// TwinCAT 3 PLC project Untitled1
// ProgramVersion: 3.1.0.8
// libraries:
//   Indradrive Library, * (Bosch)
//   Recipe Management, 3.3.1.0 (System)
//   Standard, * (System)
//   VisuElem3DPath, 3.5.6.0 (System)
//   VisuElemMeter, 3.5.6.0 (System)
//   VisuElems, 3.5.6.10 (System)
//   VisuElemsDateTime, 3.5.6.0 (System)
//   VisuElemsSpecialControls, 3.5.6.0 (System)
//   VisuElemsWinControls, 3.5.6.0 (System)
//   VisuElemTextEditor, 3.5.6.0 (System)
//   visuinputs, 3.5.6.0 (system)
//   VisuNativeControl, 3.5.6.0 (System)
//   Tc2_IoFunctions, * (Beckhoff Automation GmbH)
//   Tc2_Standard, * (Beckhoff Automation GmbH)
//   Tc2_System, * (Beckhoff Automation GmbH)
//   Tc2_Utilities, * (Beckhoff Automation GmbH)
//   Tc3_Interfaces, * (Beckhoff Automation GmbH)
//   Tc3_Module, * (Beckhoff Automation GmbH)
// project tree:
//   DUTs/ structCylinder.TcDUT, structHBMSerialCtrl.TcDUT, structHMI.TcDUT, structIndradrive.TcDUT, structMachineCtrl.TcDUT, structMachineData.TcDUT, structMotorDirect.TcDUT, structMotorInverter.TcDUT, structRecipe.TcDUT, structStationCtrl.TcDUT, structStatistic.TcDUT, structVacuum.TcDUT
//   / GlobalTextList.TcGTLO, PlcTask.TcTTO, RecipeManager.TcRMO (not stored), Visualization Manager.TcVMO (not stored)
//   GVLs/Device/ GVL_Cylinder.TcGVL, GVL_Motor.TcGVL, GVL_Nordson.TcGVL, GVL_Servo.TcGVL, GVL_Vacuum.TcGVL
//   GVLs/IO/ GVL_Ethercat.TcGVL, GVL_IO_CO.TcGVL, GVL_IO_EL.TcGVL, GVL_IO_HOR.TcGVL, GVL_IO_ER.TcGVL, GVL_Valve_Manifold.TcGVL
//   GVLs/MC/ GVL_General.TcGVL, GVL_Auto.TcGVL, GVL_Holding.TcGVL, GVL_Origin.TcGVL, GVL_Error.TcGVL, GVL_Configuration.TcGVL, GVL_HMI.TcGVL, GVL_Status.TcGVL, GVL_Symbol_Spec.TcGVL, GVL_Timer.TcGVL
//   POUs/Collator/ CO_Cylinder_Output.TcPOU, CO_Main.TcPOU, CO_Nordson.TcPOU, CO_Servo_Output.TcPOU, CO_Motor_Output.TcPOU, CO_Timers.TcPOU, CO_TestServo.TcPOU
//   POUs/Collator/Y Pusher n Bridge/ CO_YPush_Auto.TcPOU, CO_YPush_Error.TcPOU, CO_YPush_Origin.TcPOU
//   POUs/Erector/ ER_Auto_Arm.TcPOU, ER_Auto_FixedFlap.TcPOU, ER_Error.TcPOU, ER_Glue.TcPOU, ER_Origin.TcPOU, ER_Cylinder_Output.TcPOU, ER_Main.TcPOU, ER_Motor_Output.TcPOU, ER_Servo_Output.TcPOU, ER_Timers.TcPOU, ER_Vacuum_Output.TcPOU
//   POUs/Exit/ EX_Auto.TcPOU, EX_Error.TcPOU, EX_Origin.TcPOU, EX_Main.TcPOU, EX_Motor_Output.TcPOU, EX_Cylinder_Output.TcPOU, EX_LoadCell_Output.TcPOU, EX_Servo_Output.TcPOU
//   POUs/FastTask/ CO_StkRel_Cyl_FastOutput.TcPOU, FastTask_Main.TcPOU
//   POUs/FB/ fbCalculateTotalTime.TcPOU, fbCylinderCtrl_2Station.TcPOU, fbCylinderCtrl.TcPOU, fbIndradrive.TcPOU, fbMachineCtrl.TcPOU, fbMotorInverterCtrl.TcPOU, fbVacuumPumpCtrl.TcPOU, fbOnOffDevCtrl.TcPOU, fbMotorDirectCtrl.TcPOU, fbVacuumValveCtrl.TcPOU, fcComparePos.TcPOU, fcCompareWAPos.TcPOU
//   POUs/Horizontal/ Downstream_Conveyor.TcPOU, HOR_Servo_Output.TcPOU, HOR_Auto.TcPOU, HOR_Error.TcPOU, HOR_Main.TcPOU, HOR_Motor_Output.TcPOU, HOR_Origin.TcPOU, HOR_Timers.TcPOU, Option_90Deg_Conv.TcPOU
//   POUs/MC/ Calc_McPerformance.TcPOU, Check_AutorunCond.TcPOU, Check_Ethercat.TcPOU, Guard_Door.TcPOU, Emergency_Stop.TcPOU, MAIN.TcPOU, Memory_Handling.TcPOU, Recipe_Handling.TcPOU, Statistic.TcPOU, Std_System_Out.TcPOU, TouchScreen.TcPOU, Track_and_Trace.TcPOU, WarningMsg.TcPOU
//   VISUs/FB/ Std_Cylinder_Ctrl.TcVIS, Std_OnOffDev_Ctrl.TcVIS, Std_VacuumVal_Ctrl.TcVIS, Std_BoschServo_Ctrl.TcVIS
//   VISUs/Obj_Button/ ButtonGreenInd.TcVIS
//   VISUs/Obj_Indicator/ Blue_Ind.TcVIS, Green_Ind.TcVIS, Red_Ind.TcVIS, Yellow_Ind.TcVIS
//   VISUs/Obj_Switch/ ToggleSwitch1.TcVIS
//   VISUs/Prog/ IO_Monitor.TcVIS, MANUAL_STEP.TcVIS, resetbtn.TcVIS, Std_NewPassWord.TcVIS, Std_Password.TcVIS
// real-time tasks:
//   TASK PlcTask: cycle T#10ms, priority 20, ADS port 350
// I/O:
//   DEVICE Device 1 (EtherCAT), AmsNetId 169.254.27.43.2.1
//     EractorRemoteIO (EK1101) [EK1101 EtherCAT Coupler (2A E-Bus, ID switch)]
//       41DI1 (EL1809) [EL1809 16Ch. Dig. Input 24V, 3ms]
//       41DI2 (EL1809) [EL1809 16Ch. Dig. Input 24V, 3ms]
//       41DO1 (EL2809) [EL2809 16Ch. Dig. Output 24V, 0.5A]
//       41DO2 (EL2809) [EL2809 16Ch. Dig. Output 24V, 0.5A]
//       41PO1 (EL9510) [EL9510 Power supply terminal 10V] (disabled)
//       41AI1 (EL3356) [EL3356 1Ch. Ana. Input Resistor Bridge Terminal, 16bit, High Precision] (disabled)
//       41BC2 (EK1122) [EK1122 2 port EtherCAT junction]
//         EractorArmLeftValveBlock (CTEU-EtherCAT 16Byte) [CTEU-EtherCAT Fieldbus module 16Byte fix]
//         60A1 (EP1008-0001) [EP1008-0001 8 Ch. Dig. Input 24V, 3ms, M8]
//         61A1 (EP1008-0001) [EP1008-0001 8 Ch. Dig. Input 24V, 3ms, M8]
//         62A1 (EP1008-0001) [EP1008-0001 8 Ch. Dig. Input 24V, 3ms, M8]
//         66A1 (EP1008-0001) [EP1008-0001 8 Ch. Dig. Input 24V, 3ms, M8]
//         EractorArm (IndraDrive MPB16/17) [IndraDrive MPB16/17]
//         Eractor Main WA (IndraDrive MPB16/17) [IndraDrive MPB16/17]
//         Eractor HeightL WA (IndraDrive MPB16/17) [IndraDrive MPB16/17]
//         Eractor HeightR WA (IndraDrive MPB16/17) [IndraDrive MPB16/17]
//       41BC3 (EK1122) [EK1122 2 port EtherCAT junction]
//         241BC1 CollactorRemoteIO (EK1101) [EK1101 EtherCAT Coupler (2A E-Bus, ID switch)]
//           241DI1 (EL1809) [EL1809 16Ch. Dig. Input 24V, 3ms]
//           241DI2 (EL1809) [EL1809 16Ch. Dig. Input 24V, 3ms]
//           241DO1 (EL2809) [EL2809 16Ch. Dig. Output 24V, 0.5A]
//           241DO2 (EL2809) [EL2809 16Ch. Dig. Output 24V, 0.5A]
//           241BC2 (EK1122) [EK1122 2 port EtherCAT junction]
//             270A1 (CTEU-EtherCAT 16Byte) [CTEU-EtherCAT Fieldbus module 16Byte fix]
//             263A1 (EP1008-0001) [EP1008-0001 8 Ch. Dig. Input 24V, 3ms, M8]
//             264A1 (EP1008-0001) [EP1008-0001 8 Ch. Dig. Input 24V, 3ms, M8]
//             262A1 (EP1008-0001) [EP1008-0001 8 Ch. Dig. Input 24V, 3ms, M8]
//             265A1 (EP1008-0001) [EP1008-0001 8 Ch. Dig. Input 24V, 3ms, M8]
//             Tilter (IndraDrive MPB16/17) [IndraDrive MPB16/17]
//             YPusher (IndraDrive MPB16/17) [IndraDrive MPB16/17]
//         260A1 (EP1008-0001) [EP1008-0001 8 Ch. Dig. Input 24V, 3ms, M8]
//     EractorArmRightValveBlock (CTEU-EtherCAT 16Byte) [CTEU-EtherCAT Fieldbus module 16Byte fix]
//     63A1 (EP1008-0001) [EP1008-0001 8 Ch. Dig. Input 24V, 3ms, M8]
//     64A1 (EP1008-0001) [EP1008-0001 8 Ch. Dig. Input 24V, 3ms, M8]
//     65A1 (EP1008-0001) [EP1008-0001 8 Ch. Dig. Input 24V, 3ms, M8]
// variable links:
//   Untitled1/Untitled1 Instance <-> Device 1 (EtherCAT)/63A1 (EP1008-0001)
//     PlcTask Inputs/GVL_Ethercat.I_ECat_63A1 <-> InfoData/State
//     PlcTask Inputs/GVL_IO_ER.I_ER_BFlapR_Bwd <-> Channel 8/Input
//     PlcTask Inputs/GVL_IO_ER.I_ER_BFlapR_Fwd <-> Channel 7/Input
//     PlcTask Inputs/GVL_IO_ER.I_ER_BufferR_PE <-> Channel 1/Input
//     PlcTask Inputs/GVL_IO_ER.I_ER_EmptyR_PE <-> Channel 2/Input
//     PlcTask Inputs/GVL_IO_ER.I_ER_FFlapR_Bwd <-> Channel 6/Input
//     PlcTask Inputs/GVL_IO_ER.I_ER_FFlapR_Fwd <-> Channel 5/Input
//     PlcTask Inputs/GVL_IO_ER.I_EX_StpR_Dn <-> Channel 4/Input
//   Untitled1/Untitled1 Instance <-> Device 1 (EtherCAT)/64A1 (EP1008-0001)
//     PlcTask Inputs/GVL_Ethercat.I_ECat_64A1 <-> InfoData/State
//     PlcTask Inputs/GVL_IO_ER.I_ER_BFlapR_VacSw <-> Channel 7/Input
//     PlcTask Inputs/GVL_IO_ER.I_ER_CaseGuideR_Bwd <-> Channel 4/Input
//     PlcTask Inputs/GVL_IO_ER.I_ER_CaseGuideR_Fwd <-> Channel 3/Input
//     PlcTask Inputs/GVL_IO_ER.I_ER_RFlapR_Bwd <-> Channel 6/Input
//     PlcTask Inputs/GVL_IO_ER.I_ER_RFlapR_Fwd <-> Channel 5/Input
//     PlcTask Inputs/GVL_IO_ER.I_ER_StpR_Ctn_PE <-> Channel 8/Input
//     PlcTask Inputs/GVL_IO_ER.I_ER_StpR_Dn <-> Channel 2/Input
//     PlcTask Inputs/GVL_IO_ER.I_ER_StpR_Up <-> Channel 1/Input
//   Untitled1/Untitled1 Instance <-> Device 1 (EtherCAT)/65A1 (EP1008-0001)
//     PlcTask Inputs/GVL_Ethercat.I_ECat_65A1 <-> InfoData/State
//     PlcTask Inputs/GVL_IO_ER.I_ER_FlapHoldR_Bwd <-> Channel 6/Input
//     PlcTask Inputs/GVL_IO_ER.I_ER_FlapHoldR_Fwd <-> Channel 5/Input
//     PlcTask Inputs/GVL_IO_ER.I_ER_TFlapClsR_Bwd <-> Channel 4/Input
//     PlcTask Inputs/GVL_IO_ER.I_ER_TFlapClsR_Fwd <-> Channel 3/Input
//     PlcTask Inputs/GVL_IO_ER.I_ER_TFlapOpnR_Bwd <-> Channel 2/Input
//     PlcTask Inputs/GVL_IO_ER.I_ER_TFlapOpnR_Fwd <-> Channel 1/Input
//     PlcTask Inputs/GVL_IO_ER.I_EX_SquarenessR_Bwd <-> Channel 8/Input
//     PlcTask Inputs/GVL_IO_ER.I_EX_SquarenessR_Fwd <-> Channel 7/Input
//   Untitled1/Untitled1 Instance <-> Device 1 (EtherCAT)/EractorArmRightValveBlock (CTEU-EtherCAT 16Byte)
//     PlcTask Inputs/GVL_Ethercat.I_ECat_71A1 <-> InfoData/State
//     PlcTask Outputs/GVL_Valve_Manifold.QW_71A1_{1..4} <-> Outputs/QB{0..3}  (4 links)
//   Untitled1/Untitled1 Instance <-> Device 1 (EtherCAT)/EractorRemoteIO (EK1101)
//     PlcTask Inputs/GVL_Ethercat.I_ECat_41BC1 <-> InfoData/State
//   Untitled1/Untitled1 Instance <-> Device 1 (EtherCAT)/EractorRemoteIO (EK1101)/41AI1 (EL3356)
//     PlcTask Inputs/GVL_IO_ER.I_Weighing <-> RMB Value (INT32)/Value
//     PlcTask Inputs/GVL_IO_ER.I_Weighing_Status_SteadyBit <-> RMB Status/Status/Steady state
//   Untitled1/Untitled1 Instance <-> Device 1 (EtherCAT)/EractorRemoteIO (EK1101)/41BC2 (EK1122)
//     PlcTask Inputs/GVL_Ethercat.I_ECat_41BC2 <-> InfoData/State
//   Untitled1/Untitled1 Instance <-> Device 1 (EtherCAT)/EractorRemoteIO (EK1101)/41BC2 (EK1122)/60A1 (EP1008-0001)
//     PlcTask Inputs/GVL_Ethercat.I_ECat_60A1 <-> InfoData/State
//     PlcTask Inputs/GVL_IO_ER.I_ER_BFlapL_Bwd <-> Channel 8/Input
//     PlcTask Inputs/GVL_IO_ER.I_ER_BFlapL_Fwd <-> Channel 7/Input
//     PlcTask Inputs/GVL_IO_ER.I_ER_BufferL_PE <-> Channel 1/Input
//     PlcTask Inputs/GVL_IO_ER.I_ER_EmptyL_PE <-> Channel 2/Input
//     PlcTask Inputs/GVL_IO_ER.I_ER_FFlapL_Bwd <-> Channel 6/Input
//     PlcTask Inputs/GVL_IO_ER.I_ER_FFlapL_Fwd <-> Channel 5/Input
//     PlcTask Inputs/GVL_IO_ER.I_ER_RefillL_PE <-> Channel 3/Input
//     PlcTask Inputs/GVL_IO_ER.I_EX_StpL_Dn <-> Channel 4/Input
//   Untitled1/Untitled1 Instance <-> Device 1 (EtherCAT)/EractorRemoteIO (EK1101)/41BC2 (EK1122)/61A1 (EP1008-0001)
//     PlcTask Inputs/GVL_Ethercat.I_ECat_61A1 <-> InfoData/State
//     PlcTask Inputs/GVL_IO_ER.I_ER_BFlapL_VacSw <-> Channel 7/Input
//     PlcTask Inputs/GVL_IO_ER.I_ER_CaseGuideL_Bwd <-> Channel 4/Input
//     PlcTask Inputs/GVL_IO_ER.I_ER_CaseGuideL_Fwd <-> Channel 3/Input
//     PlcTask Inputs/GVL_IO_ER.I_ER_RFlapL_Bwd <-> Channel 6/Input
//     PlcTask Inputs/GVL_IO_ER.I_ER_RFlapL_Fwd <-> Channel 5/Input
//     PlcTask Inputs/GVL_IO_ER.I_ER_StpL_Ctn_PE <-> Channel 8/Input
//     PlcTask Inputs/GVL_IO_ER.I_ER_StpL_Dn <-> Channel 2/Input
//     PlcTask Inputs/GVL_IO_ER.I_ER_StpL_Up <-> Channel 1/Input
//   Untitled1/Untitled1 Instance <-> Device 1 (EtherCAT)/EractorRemoteIO (EK1101)/41BC2 (EK1122)/62A1 (EP1008-0001)
//     PlcTask Inputs/GVL_Ethercat.I_ECat_62A1 <-> InfoData/State
//     PlcTask Inputs/GVL_IO_ER.I_ER_FlapHoldL_Bwd <-> Channel 6/Input
//     PlcTask Inputs/GVL_IO_ER.I_ER_FlapHoldL_Fwd <-> Channel 5/Input
//     PlcTask Inputs/GVL_IO_ER.I_ER_TFlapClsL_Bwd <-> Channel 4/Input
//     PlcTask Inputs/GVL_IO_ER.I_ER_TFlapClsL_Fwd <-> Channel 3/Input
//     PlcTask Inputs/GVL_IO_ER.I_ER_TFlapOpnL_Bwd <-> Channel 2/Input
//     PlcTask Inputs/GVL_IO_ER.I_ER_TFlapOpnL_Fwd <-> Channel 1/Input
//     PlcTask Inputs/GVL_IO_ER.I_EX_SquarenessL_Bwd <-> Channel 8/Input
//     PlcTask Inputs/GVL_IO_ER.I_EX_SquarenessL_Fwd <-> Channel 7/Input
//   Untitled1/Untitled1 Instance <-> Device 1 (EtherCAT)/EractorRemoteIO (EK1101)/41BC2 (EK1122)/66A1 (EP1008-0001)
//     PlcTask Inputs/GVL_Ethercat.I_ECat_66A1 <-> InfoData/State
//     PlcTask Inputs/GVL_IO_ER.I_ER_ArmTilt_Bwd <-> Channel 2/Input
//     PlcTask Inputs/GVL_IO_ER.I_ER_ArmTilt_Fwd <-> Channel 1/Input
//     PlcTask Inputs/GVL_IO_ER.I_ER_Arm_Dn <-> Channel 4/Input
//     PlcTask Inputs/GVL_IO_ER.I_ER_Arm_Up <-> Channel 3/Input
//     PlcTask Inputs/GVL_IO_ER.I_ER_Arm_VacSw <-> Channel 7/Input
//     PlcTask Inputs/GVL_IO_ER.I_EX_Cv_Ctn_PE <-> Channel 8/Input
//   Untitled1/Untitled1 Instance <-> Device 1 (EtherCAT)/EractorRemoteIO (EK1101)/41BC2 (EK1122)/Eractor HeightL WA (IndraDrive MPB16/17)
//     PlcTask Inputs/GVL_Servo.EX_HeightL_WA_Srv_Input/diIstgeschwindigkeit <-> AT/Velocity feedback value
//     PlcTask Inputs/GVL_Servo.EX_HeightL_WA_Srv_Input/diLageistwert <-> AT/Active position feedback value
//     PlcTask Inputs/GVL_Servo.EX_HeightL_WA_Srv_Input/dwDiagnosenummer <-> AT/Diagnostic message number
//     PlcTask Inputs/GVL_Servo.EX_HeightL_WA_Srv_Input/wAntriebsstatuswort <-> AT/Drive status word
//     PlcTask Inputs/GVL_Servo.EX_HeightL_WA_Srv_Input/wSignalstatuswort <-> AT/Signal status word
//     PlcTask Inputs/GVL_Servo.EX_HeightL_WA_Srv_State <-> InfoData/State
//     PlcTask Outputs/GVL_Servo.EX_HeightL_WA_Srv_Feedrate <-> MDT/Feedrate override
//     PlcTask Outputs/GVL_Servo.EX_HeightL_WA_Srv_Output/diPositioniergeschwindigkeit <-> MDT/Positioning velocity
//     PlcTask Outputs/GVL_Servo.EX_HeightL_WA_Srv_Output/diPositioniersollwert <-> MDT/Positioning command value
//     PlcTask Outputs/GVL_Servo.EX_HeightL_WA_Srv_Output/wMastersteuerwort <-> MDT/Master control word
//     PlcTask Outputs/GVL_Servo.EX_HeightL_WA_Srv_Output/wSignalsteuerwort <-> MDT/Signal control word
//   Untitled1/Untitled1 Instance <-> Device 1 (EtherCAT)/EractorRemoteIO (EK1101)/41BC2 (EK1122)/Eractor HeightR WA (IndraDrive MPB16/17)
//     PlcTask Inputs/GVL_Servo.EX_HeightR_WA_Srv_Input/diIstgeschwindigkeit <-> AT/Velocity feedback value
//     PlcTask Inputs/GVL_Servo.EX_HeightR_WA_Srv_Input/diLageistwert <-> AT/Active position feedback value
//     PlcTask Inputs/GVL_Servo.EX_HeightR_WA_Srv_Input/dwDiagnosenummer <-> AT/Diagnostic message number
//     PlcTask Inputs/GVL_Servo.EX_HeightR_WA_Srv_Input/wAntriebsstatuswort <-> AT/Drive status word
//     PlcTask Inputs/GVL_Servo.EX_HeightR_WA_Srv_Input/wSignalstatuswort <-> AT/Signal status word
//     PlcTask Inputs/GVL_Servo.EX_HeightR_WA_Srv_State <-> InfoData/State
//     PlcTask Outputs/GVL_Servo.EX_HeightR_WA_Srv_Feedrate <-> MDT/Feedrate override
//     PlcTask Outputs/GVL_Servo.EX_HeightR_WA_Srv_Output/diPositioniergeschwindigkeit <-> MDT/Positioning velocity
//     PlcTask Outputs/GVL_Servo.EX_HeightR_WA_Srv_Output/diPositioniersollwert <-> MDT/Positioning command value
//     PlcTask Outputs/GVL_Servo.EX_HeightR_WA_Srv_Output/wMastersteuerwort <-> MDT/Master control word
//     PlcTask Outputs/GVL_Servo.EX_HeightR_WA_Srv_Output/wSignalsteuerwort <-> MDT/Signal control word
//   Untitled1/Untitled1 Instance <-> Device 1 (EtherCAT)/EractorRemoteIO (EK1101)/41BC2 (EK1122)/Eractor Main WA (IndraDrive MPB16/17)
//     PlcTask Inputs/GVL_Servo.ER_WA_Srv_Input/diIstgeschwindigkeit <-> AT/Geschwindigkeits-Istwert
//     PlcTask Inputs/GVL_Servo.ER_WA_Srv_Input/diLageistwert <-> AT/Aktiver Lageistwert
//     PlcTask Inputs/GVL_Servo.ER_WA_Srv_Input/dwDiagnosenummer <-> AT/Diagnose-Nummer
//     PlcTask Inputs/GVL_Servo.ER_WA_Srv_Input/wAntriebsstatuswort <-> AT/Drive status word
//     PlcTask Inputs/GVL_Servo.ER_WA_Srv_Input/wSignalstatuswort <-> AT/Signal-Statuswort
//     PlcTask Inputs/GVL_Servo.ER_WA_Srv_State <-> InfoData/State
//     PlcTask Outputs/GVL_Servo.ER_WA_Srv_Feedrate <-> MDT/Feedrate-Override
//     PlcTask Outputs/GVL_Servo.ER_WA_Srv_Output/diPositioniergeschwindigkeit <-> MDT/Positioniergeschwindigkeit
//     PlcTask Outputs/GVL_Servo.ER_WA_Srv_Output/diPositioniersollwert <-> MDT/Positioniersollwert
//     PlcTask Outputs/GVL_Servo.ER_WA_Srv_Output/wMastersteuerwort <-> MDT/Master control word
//     PlcTask Outputs/GVL_Servo.ER_WA_Srv_Output/wSignalsteuerwort <-> MDT/Signal-Steuerwort
//   Untitled1/Untitled1 Instance <-> Device 1 (EtherCAT)/EractorRemoteIO (EK1101)/41BC2 (EK1122)/EractorArm (IndraDrive MPB16/17)
//     PlcTask Inputs/GVL_Servo.ER_Arm_Srv_Input/diIstgeschwindigkeit <-> AT/Velocity feedback value
//     PlcTask Inputs/GVL_Servo.ER_Arm_Srv_Input/diLageistwert <-> AT/Active position feedback value
//     PlcTask Inputs/GVL_Servo.ER_Arm_Srv_Input/dwDiagnosenummer <-> AT/Diagnostic message number
//     PlcTask Inputs/GVL_Servo.ER_Arm_Srv_Input/wAntriebsstatuswort <-> AT/Drive status word
//     PlcTask Inputs/GVL_Servo.ER_Arm_Srv_Input/wSignalstatuswort <-> AT/Signal status word
//     PlcTask Inputs/GVL_Servo.ER_Arm_Srv_State <-> InfoData/State
//     PlcTask Outputs/GVL_Servo.ER_Arm_Srv_Feedrate <-> MDT/Feedrate override
//     PlcTask Outputs/GVL_Servo.ER_Arm_Srv_Output/diPositioniergeschwindigkeit <-> MDT/Positioning velocity
//     PlcTask Outputs/GVL_Servo.ER_Arm_Srv_Output/diPositioniersollwert <-> MDT/Positioning command value
//     PlcTask Outputs/GVL_Servo.ER_Arm_Srv_Output/wMastersteuerwort <-> MDT/Master control word
//     PlcTask Outputs/GVL_Servo.ER_Arm_Srv_Output/wSignalsteuerwort <-> MDT/Signal control word
//   Untitled1/Untitled1 Instance <-> Device 1 (EtherCAT)/EractorRemoteIO (EK1101)/41BC2 (EK1122)/EractorArmLeftValveBlock (CTEU-EtherCAT 16Byte)
//     PlcTask Inputs/GVL_Ethercat.I_ECat_70A1 <-> InfoData/State
//     PlcTask Outputs/GVL_Valve_Manifold.QW_70A1_{1..4} <-> Outputs/QB{0..3}  (4 links)
//   Untitled1/Untitled1 Instance <-> Device 1 (EtherCAT)/EractorRemoteIO (EK1101)/41BC3 (EK1122)
//     PlcTask Inputs/GVL_Ethercat.I_ECat_41BC3 <-> InfoData/State
//   Untitled1/Untitled1 Instance <-> Device 1 (EtherCAT)/EractorRemoteIO (EK1101)/41BC3 (EK1122)/241BC1 CollactorRemoteIO (EK1101)
//     PlcTask Inputs/GVL_Ethercat.I_ECat_141BC1 <-> InfoData/State
//   Untitled1/Untitled1 Instance <-> Device 1 (EtherCAT)/EractorRemoteIO (EK1101)/41BC3 (EK1122)/241BC1 CollactorRemoteIO (EK1101)/241BC2 (EK1122)
//     PlcTask Inputs/GVL_Ethercat.I_ECat_141BC2 <-> InfoData/State
//   Untitled1/Untitled1 Instance <-> Device 1 (EtherCAT)/EractorRemoteIO (EK1101)/41BC3 (EK1122)/241BC1 CollactorRemoteIO (EK1101)/241BC2 (EK1122)/262A1 (EP1008-0001)
//     PlcTask Inputs/GVL_Ethercat.I_ECat_162A1 <-> InfoData/State
//     PlcTask Inputs/GVL_IO_CO.I_CO_YPush_Dn <-> Channel 2/Input
//     PlcTask Inputs/GVL_IO_CO.I_CO_YPush_Strk_Bwd <-> Channel 4/Input
//     PlcTask Inputs/GVL_IO_CO.I_CO_YPush_Strk_Fwd <-> Channel 3/Input
//     PlcTask Inputs/GVL_IO_CO.I_CO_YPush_Up <-> Channel 1/Input
//   Untitled1/Untitled1 Instance <-> Device 1 (EtherCAT)/EractorRemoteIO (EK1101)/41BC3 (EK1122)/241BC1 CollactorRemoteIO (EK1101)/241BC2 (EK1122)/263A1 (EP1008-0001)
//     PlcTask Inputs/GVL_Ethercat.I_ECat_160A1 <-> InfoData/State
//     PlcTask Inputs/GVL_IO_CO.I_CO_Brdg_Bwd <-> Channel 6/Input
//     PlcTask Inputs/GVL_IO_CO.I_CO_Brdg_Fwd <-> Channel 5/Input
//     PlcTask Inputs/GVL_IO_CO.I_CO_FFlapGuide_Bwd <-> Channel 2/Input
//     PlcTask Inputs/GVL_IO_CO.I_CO_FFlapGuide_Fwd <-> Channel 1/Input
//     PlcTask Inputs/GVL_IO_CO.I_CO_PalletInPosition <-> Channel 7/Input
//     PlcTask Inputs/GVL_IO_CO.I_CO_RFlapGuide_Bwd <-> Channel 4/Input
//     PlcTask Inputs/GVL_IO_CO.I_CO_RFlapGuide_Fwd <-> Channel 3/Input
//   Untitled1/Untitled1 Instance <-> Device 1 (EtherCAT)/EractorRemoteIO (EK1101)/41BC3 (EK1122)/241BC1 CollactorRemoteIO (EK1101)/241BC2 (EK1122)/264A1 (EP1008-0001)
//     PlcTask Inputs/GVL_Ethercat.I_ECat_161A1 <-> InfoData/State
//     PlcTask Inputs/GVL_IO_CO.I_CO_PalletLocating_Bwd <-> Channel 6/Input
//     PlcTask Inputs/GVL_IO_CO.I_CO_PalletLocating_Fwd <-> Channel 5/Input
//     PlcTask Inputs/GVL_IO_CO.I_CO_Sing1_Bwd <-> Channel 2/Input
//     PlcTask Inputs/GVL_IO_CO.I_CO_Sing2_Bwd <-> Channel 4/Input
//     PlcTask Inputs/GVL_IO_CO.I_CO_Sing1_Fwd <-> Channel 1/Input
//     PlcTask Inputs/GVL_IO_CO.I_CO_Sing2_Fwd <-> Channel 3/Input
//   Untitled1/Untitled1 Instance <-> Device 1 (EtherCAT)/EractorRemoteIO (EK1101)/41BC3 (EK1122)/241BC1 CollactorRemoteIO (EK1101)/241BC2 (EK1122)/265A1 (EP1008-0001)
//     PlcTask Inputs/GVL_IO_CO.I_CO_Bdl_PE{1..6} <-> Channel {1..6}/Input  (6 links)
//   Untitled1/Untitled1 Instance <-> Device 1 (EtherCAT)/EractorRemoteIO (EK1101)/41BC3 (EK1122)/241BC1 CollactorRemoteIO (EK1101)/241BC2 (EK1122)/270A1 (CTEU-EtherCAT 16Byte)
//     PlcTask Inputs/GVL_Ethercat.I_ECat_170A1 <-> InfoData/State
//     PlcTask Outputs/GVL_Valve_Manifold.QW_170A1_1 <-> RxPDO/Output 1
//     PlcTask Outputs/GVL_Valve_Manifold.QW_170A1_2 <-> RxPDO/Output 2
//   Untitled1/Untitled1 Instance <-> Device 1 (EtherCAT)/EractorRemoteIO (EK1101)/41BC3 (EK1122)/241BC1 CollactorRemoteIO (EK1101)/241BC2 (EK1122)/Tilter (IndraDrive MPB16/17)
//     PlcTask Inputs/GVL_Servo.EX_Tilt_Srv_Input/diIstgeschwindigkeit <-> AT/Geschwindigkeits-Istwert
//     PlcTask Inputs/GVL_Servo.EX_Tilt_Srv_Input/diLageistwert <-> AT/Aktiver Lageistwert
//     PlcTask Inputs/GVL_Servo.EX_Tilt_Srv_Input/dwDiagnosenummer <-> AT/Diagnose-Nummer
//     PlcTask Inputs/GVL_Servo.EX_Tilt_Srv_Input/wAntriebsstatuswort <-> AT/Drive status word
//     PlcTask Inputs/GVL_Servo.EX_Tilt_Srv_Input/wSignalstatuswort <-> AT/Signal-Statuswort
//     PlcTask Inputs/GVL_Servo.EX_Tilt_Srv_State <-> InfoData/State
//     PlcTask Outputs/GVL_Servo.EX_Tilt_Srv_Feedrate <-> MDT/Feedrate-Override
//     PlcTask Outputs/GVL_Servo.EX_Tilt_Srv_Output/diPositioniergeschwindigkeit <-> MDT/Positioniergeschwindigkeit
//     PlcTask Outputs/GVL_Servo.EX_Tilt_Srv_Output/diPositioniersollwert <-> MDT/Positioniersollwert
//     PlcTask Outputs/GVL_Servo.EX_Tilt_Srv_Output/wMastersteuerwort <-> MDT/Master control word
//     PlcTask Outputs/GVL_Servo.EX_Tilt_Srv_Output/wSignalsteuerwort <-> MDT/Signal-Steuerwort
//   Untitled1/Untitled1 Instance <-> Device 1 (EtherCAT)/EractorRemoteIO (EK1101)/41BC3 (EK1122)/241BC1 CollactorRemoteIO (EK1101)/241BC2 (EK1122)/YPusher (IndraDrive MPB16/17)
//     PlcTask Inputs/GVL_Servo.CO_YPush_Srv_Input/diIstgeschwindigkeit <-> AT/Geschwindigkeits-Istwert
//     PlcTask Inputs/GVL_Servo.CO_YPush_Srv_Input/diLageistwert <-> AT/Aktiver Lageistwert
//     PlcTask Inputs/GVL_Servo.CO_YPush_Srv_Input/dwDiagnosenummer <-> AT/Diagnose-Nummer
//     PlcTask Inputs/GVL_Servo.CO_YPush_Srv_Input/wAntriebsstatuswort <-> AT/Drive status word
//     PlcTask Inputs/GVL_Servo.CO_YPush_Srv_Input/wSignalstatuswort <-> AT/Signal-Statuswort
//     PlcTask Inputs/GVL_Servo.CO_YPush_Srv_State <-> InfoData/State
//     PlcTask Outputs/GVL_Servo.CO_YPush_Srv_Feedrate <-> MDT/Feedrate-Override
//     PlcTask Outputs/GVL_Servo.CO_YPush_Srv_Output/diPositioniergeschwindigkeit <-> MDT/Positioniergeschwindigkeit
//     PlcTask Outputs/GVL_Servo.CO_YPush_Srv_Output/diPositioniersollwert <-> MDT/Positioniersollwert
//     PlcTask Outputs/GVL_Servo.CO_YPush_Srv_Output/wMastersteuerwort <-> MDT/Master control word
//     PlcTask Outputs/GVL_Servo.CO_YPush_Srv_Output/wSignalsteuerwort <-> MDT/Signal-Steuerwort
//   Untitled1/Untitled1 Instance <-> Device 1 (EtherCAT)/EractorRemoteIO (EK1101)/41BC3 (EK1122)/241BC1 CollactorRemoteIO (EK1101)/241DI1 (EL1809)
//     PlcTask Inputs/GVL_Ethercat.I_ECat_141DI1 <-> InfoData/State
//     PlcTask Inputs/GVL_IO_CO.I_CO_Cv_InvRdy <-> Channel 12/Input
//     PlcTask Inputs/GVL_IO_CO.I_Nord_Alm <-> Channel 10/Input
//     PlcTask Inputs/GVL_IO_CO.I_Nord_Rdy <-> Channel 9/Input
//     PlcTask Inputs/GVL_IO_CO.I_Nord_TankLow <-> Channel 11/Input
//     PlcTask Inputs/GVL_IO_CO.I_PressSw_OK <-> Channel 15/Input
//     PlcTask Inputs/GVL_IO_HOR.I_CO_PusherReady <-> Channel 7/Input
//     PlcTask Inputs/GVL_IO_HOR.I_EStop_Collator <-> Channel 8/Input
//     PlcTask Inputs/GVL_IO_HOR.I_EStop_HorExit <-> Channel 6/Input
//     PlcTask Inputs/GVL_IO_HOR.I_EStop_HorL <-> Channel 4/Input
//     PlcTask Inputs/GVL_IO_HOR.I_EStop_HorR <-> Channel 5/Input
//     PlcTask Inputs/GVL_IO_HOR.I_HLC_SC_OK <-> Channel 3/Input
//     PlcTask Inputs/GVL_IO_HOR.I_HOR_BotCv_InvRdy <-> Channel 2/Input
//     PlcTask Inputs/GVL_IO_HOR.I_HOR_TopCv_InvRdy <-> Channel 1/Input
//   Untitled1/Untitled1 Instance <-> Device 1 (EtherCAT)/EractorRemoteIO (EK1101)/41BC3 (EK1122)/241BC1 CollactorRemoteIO (EK1101)/241DI2 (EL1809)
//     PlcTask Inputs/GVL_IO_CO.I_COL_Front_Door_Sen <-> Channel 3/Input
//     PlcTask Inputs/GVL_IO_CO.I_COL_Rear_Door_Sen <-> Channel 4/Input
//     PlcTask Inputs/GVL_IO_CO.I_Pneumatic_Sup1_ON <-> Channel 1/Input
//     PlcTask Inputs/GVL_IO_CO.I_Pneumatic_Sup2_ON <-> Channel 2/Input
//   Untitled1/Untitled1 Instance <-> Device 1 (EtherCAT)/EractorRemoteIO (EK1101)/41BC3 (EK1122)/241BC1 CollactorRemoteIO (EK1101)/241DO1 (EL2809)
//     PlcTask Inputs/GVL_Ethercat.I_ECat_141DO1 <-> InfoData/State
//     PlcTask Outputs/GVL_IO_HOR.O_HOR_BotCv_Mtr_Dirc <-> Channel 14/Output
//     PlcTask Outputs/GVL_IO_HOR.O_HOR_BotCv_Mtr_Run <-> Channel 13/Output
//     PlcTask Outputs/GVL_IO_HOR.O_HOR_BotCv_Mtr_Spd1 <-> Channel 15/Output
//     PlcTask Outputs/GVL_IO_HOR.O_HOR_BotCv_Mtr_Spd2 <-> Channel 16/Output
//     PlcTask Outputs/GVL_IO_HOR.O_HOR_LC_Mute1 <-> Channel 2/Output
//     PlcTask Outputs/GVL_IO_HOR.O_HOR_LC_Mute2 <-> Channel 3/Output
//     PlcTask Outputs/GVL_IO_HOR.O_HOR_TiltCV1_On <-> Channel 4/Output
//     PlcTask Outputs/GVL_IO_HOR.O_HOR_TiltCV2_On <-> Channel 5/Output
//     PlcTask Outputs/GVL_IO_HOR.O_HOR_TopCv_Mtr_Dirc <-> Channel 10/Output
//     PlcTask Outputs/GVL_IO_HOR.O_HOR_TopCv_Mtr_Run <-> Channel 9/Output
//     PlcTask Outputs/GVL_IO_HOR.O_HOR_TopCv_Mtr_Spd1 <-> Channel 11/Output
//     PlcTask Outputs/GVL_IO_HOR.O_HOR_TopCv_Mtr_Spd2 <-> Channel 12/Output
//   Untitled1/Untitled1 Instance <-> Device 1 (EtherCAT)/EractorRemoteIO (EK1101)/41BC3 (EK1122)/241BC1 CollactorRemoteIO (EK1101)/241DO2 (EL2809)
//     PlcTask Inputs/GVL_IO_CO.IW_141DI1 <-> InfoData/State
//     PlcTask Outputs/GVL_IO_CO.O_Nord_Auto <-> Channel 1/Output
//     PlcTask Outputs/GVL_IO_CO.O_Nord_HeaterOn <-> Channel 3/Output
//     PlcTask Outputs/GVL_IO_CO.O_Nord_Standby <-> Channel 2/Output
//   Untitled1/Untitled1 Instance <-> Device 1 (EtherCAT)/EractorRemoteIO (EK1101)/41BC3 (EK1122)/260A1 (EP1008-0001)
//     PlcTask Inputs/GVL_Ethercat.I_ECat_260A1 <-> InfoData/State
//     PlcTask Inputs/GVL_IO_HOR.I_HOR_DnStream_Cv_Full <-> Channel 4/Input
//     PlcTask Inputs/GVL_IO_HOR.I_HOR_Entry_Cv_Present <-> Channel 1/Input
//     PlcTask Inputs/GVL_IO_HOR.I_HOR_Left_Door <-> Channel 5/Input
//     PlcTask Inputs/GVL_IO_HOR.I_HOR_Right_Door <-> Channel 6/Input
//     PlcTask Inputs/GVL_IO_HOR.I_HOR_TapeL_Empty_PE <-> Channel 7/Input
//     PlcTask Inputs/GVL_IO_HOR.I_HOR_TapeL_Present_PE <-> Channel 2/Input
//     PlcTask Inputs/GVL_IO_HOR.I_HOR_TapeR_Empty_PE <-> Channel 8/Input
//     PlcTask Inputs/GVL_IO_HOR.I_HOR_TapeR_Present_PE <-> Channel 3/Input
//   Untitled1/Untitled1 Instance <-> Device 1 (EtherCAT)/EractorRemoteIO (EK1101)/41DI1 (EL1809)
//     PlcTask Inputs/GVL_Ethercat.I_ECat_41DI1 <-> InfoData/State
//     PlcTask Inputs/GVL_IO_ER.I_CartonCV_M1M2_OK <-> Channel 9/Input
//     PlcTask Inputs/GVL_IO_ER.I_Case_Infeed_Safety_Ok <-> Channel 7/Input
//     PlcTask Inputs/GVL_IO_ER.I_Door_SC_OK <-> Channel 6/Input
//     PlcTask Inputs/GVL_IO_ER.I_Emg_SC_OK <-> Channel 5/Input
//     PlcTask Inputs/GVL_IO_ER.I_Erector_Front_Door_Sen <-> Channel 12/Input
//     PlcTask Inputs/GVL_IO_ER.I_IncomingPowerPhase_OK <-> Channel 11/Input
//     PlcTask Inputs/GVL_IO_ER.I_PCUPS_OK <-> Channel 8/Input
//     PlcTask Inputs/GVL_IO_ER.I_Reset_PB <-> Channel 3/Input
//     PlcTask Inputs/GVL_IO_ER.I_Safety_OK <-> Channel 4/Input
//     PlcTask Inputs/GVL_IO_ER.I_Start_PB <-> Channel 1/Input
//     PlcTask Inputs/GVL_IO_ER.I_Stop_PB <-> Channel 2/Input
//     PlcTask Inputs/GVL_IO_ER.I_Weighing_CV_OK <-> Channel 10/Input
//     PlcTask Inputs/GVL_IO_ER.I_erector_Rear_Door_Sen <-> Channel 13/Input
//   Untitled1/Untitled1 Instance <-> Device 1 (EtherCAT)/EractorRemoteIO (EK1101)/41DI2 (EL1809)
//     PlcTask Inputs/GVL_Ethercat.I_ECat_41DI2 <-> InfoData/State
//     PlcTask Inputs/GVL_IO_ER.I_DnStream_ExitJam <-> Channel 5/Input
//     PlcTask Inputs/GVL_IO_ER.I_DnStream_InProd <-> Channel 6/Input
//     PlcTask Inputs/GVL_IO_ER.I_EStop_Panel <-> Channel 16/Input
//     PlcTask Inputs/GVL_IO_ER.I_TnT_Healthy <-> Channel 9/Input
//     PlcTask Inputs/GVL_IO_ER.I_TnT_LabelerINP <-> Channel 10/Input
//     PlcTask Inputs/GVL_IO_ER.I_UpStream_ExitJam <-> Channel 1/Input
//     PlcTask Inputs/GVL_IO_ER.I_UpStream_InProd <-> Channel 2/Input
//   Untitled1/Untitled1 Instance <-> Device 1 (EtherCAT)/EractorRemoteIO (EK1101)/41DO1 (EL2809)
//     PlcTask Inputs/GVL_Ethercat.I_ECat_41DO1 <-> InfoData/State
//     PlcTask Outputs/GVL_IO_ER.O_Buz_TL <-> Channel 7/Output
//     PlcTask Outputs/GVL_IO_ER.O_DoorLock <-> Channel 8/Output
//     PlcTask Outputs/GVL_IO_ER.O_ER_Arm_Vac_On <-> Channel 14/Output
//     PlcTask Outputs/GVL_IO_ER.O_ER_BFlapL_Vac_On <-> Channel 12/Output
//     PlcTask Outputs/GVL_IO_ER.O_ER_BFlapR_Vac_On <-> Channel 13/Output
//     PlcTask Outputs/GVL_IO_ER.O_ER_BufCv_Mtr1_On <-> Channel 10/Output
//     PlcTask Outputs/GVL_IO_ER.O_ER_BufCv_Mtr2_On <-> Channel 11/Output
//     PlcTask Outputs/GVL_IO_ER.O_Grn_TL <-> Channel 6/Output
//     PlcTask Outputs/GVL_IO_ER.O_Nord_ValveL_On <-> Channel 15/Output
//     PlcTask Outputs/GVL_IO_ER.O_Nord_ValveR_On <-> Channel 16/Output
//     PlcTask Outputs/GVL_IO_ER.O_Red_TL <-> Channel 4/Output
//     PlcTask Outputs/GVL_IO_ER.O_Reset_PL <-> Channel 3/Output
//     PlcTask Outputs/GVL_IO_ER.O_Start_PL <-> Channel 1/Output
//     PlcTask Outputs/GVL_IO_ER.O_Stop_PL <-> Channel 2/Output
//     PlcTask Outputs/GVL_IO_ER.O_Weighing_CV_ON <-> Channel 9/Output
//     PlcTask Outputs/GVL_IO_ER.O_Yel_TL <-> Channel 5/Output
//   Untitled1/Untitled1 Instance <-> Device 1 (EtherCAT)/EractorRemoteIO (EK1101)/41DO2 (EL2809)
//     PlcTask Inputs/GVL_Ethercat.I_ECat_41DO2 <-> InfoData/State
//     PlcTask Outputs/GVL_IO_ER.O_DnStream_Reject <-> Channel 15/Output
//     PlcTask Outputs/GVL_IO_ER.O_DnStream_ReqToStpNC <-> Channel 14/Output
//     PlcTask Outputs/GVL_IO_ER.O_DnStream_ReqToStpNO <-> Channel 13/Output
//     PlcTask Outputs/GVL_IO_ER.O_TnT_CaseFormat <-> Channel 1/Output
//     PlcTask Outputs/GVL_IO_ER.O_TnT_CaseIndex <-> Channel 4/Output
//     PlcTask Outputs/GVL_IO_ER.O_TnT_CrossPushForward <-> Channel 3/Output
//     PlcTask Outputs/GVL_IO_ER.O_TnT_CrossPushToCase <-> Channel 2/Output
//     PlcTask Outputs/GVL_IO_ER.O_TnT_GoodCaseDischarge <-> Channel 5/Output
//     PlcTask Outputs/GVL_IO_ER.O_UpStream_ReqEmptying <-> Channel 12/Output
//     PlcTask Outputs/GVL_IO_ER.O_UpStream_ReqToStpNC <-> Channel 10/Output
//     PlcTask Outputs/GVL_IO_ER.O_UpStream_ReqToStpNO <-> Channel 9/Output

CONFIGURATION Untitled1
    RESOURCE PLC ON TwinCAT3
        TASK PlcTask(INTERVAL := T#10ms, PRIORITY := 20);
        PROGRAM MAIN WITH PlcTask : MAIN;
    END_RESOURCE
END_CONFIGURATION

// ---- DUTs/structCylinder.TcDUT
TYPE structCylinder :
STRUCT
	In_CylName:STRING;
	(*Trigger*)
	T_ManWork:BOOL;
	T_ManHome:BOOL;
	In_AutoWork:BOOL;
	In_AutoHome:BOOL;
	In_OrgWork:BOOL;
	In_OrgHome:BOOL;
	(*Mechanical Interlock*)
	In_WorkXLock:BOOL;
	In_HomeXLock:BOOL;
	E_WorkErr:BOOL;
	E_HomeErr:BOOL;
	S_WorkPos:BOOL;
	S_HomePos:BOOL;

END_STRUCT
END_TYPE

// ---- DUTs/structHBMSerialCtrl.TcDUT
TYPE structHBMSerialCtrl :
STRUCT
	In_Init:BOOL;
	In_Trigger:BOOL;
	
	Out_ReceiveDone:BOOL;
	Out_WeightResult:REAL;
	Out_InitOK:BOOL;	
	Out_ErrorWord:INT;
	Out_ErrorString:STRING;

END_STRUCT
END_TYPE

// ---- DUTs/structHMI.TcDUT
TYPE structHMI :
STRUCT
	
	T_Auto: 			BOOL;
	T_Manual:			BOOL;
	T_DryRun: 			BOOL;
	T_OriginSearch:		BOOL;
	T_StationOriginSearch:BOOL;
	T_Start:			BOOL;
	T_Stop:				BOOL;
	T_Reset :			BOOL;
 	T_Station_BypassP: 	ARRAY [0..50] OF BOOL;
	T_BypassDoor: 		BOOL;
	T_BypassBuzzer:		BOOL;
	T_BuzzerOff :		BOOL;
	T_AutoMsgAlarm: 	BOOL;
	T_StatusString: 	STRING;
	T_StatusStringInt:	INT;

	T_AutoRunString:		STRING;

	T_StepRun:			BOOL;
	T_StepStop:			BOOL;
	T_StepBwd:			BOOL;
	T_StepFwd:			BOOL;
	T_StationError:		BOOL;
	T_Origin:			BOOL;
	T_OneCycleRun:		BOOL;
	T_ManualCycleTime:	TIME;
	T_Curr_Step_Station: 	UINT;
	T_EndProd:			BOOL;
	
	T_StepRunning:		BOOL;
	T_OriginRunning:	BOOL;

	V_StepRunCurrStation:	STRING;
	V_StepRunStatus:		STRING;
	V_AutorunString:		STRING;
	V_MachineSpeed:		INT;
	
	T_LoadNewRecipe:BOOL;
	T_ClearCollatorMem:BOOL;
	T_ClearBufferMem:BOOL;
	T_ClearErectorMem:BOOL;
	T_ClearElevatorMem:BOOL;
	T_ClearExitMem:BOOL;
	T_ClearAllMem:BOOL;
	
	T_ResetCounters:BOOL;
	T_ResetTotalTime:BOOL;
	
	T_PurgeErectorCase:BOOL;

END_STRUCT
END_TYPE

// ---- DUTs/structIndradrive.TcDUT
TYPE structIndradrive :
STRUCT
	In_ServoOn:BOOL;
	In_JogFwd:BOOL;
	In_JogBwd:BOOL;
	In_MoveHome:BOOL;
	In_SetAbsRef:BOOL;
	In_MoveAbs:BOOL;
	In_MoveRel:BOOL;
	In_StopMove:BOOL;
	In_VelCmd:REAL;
	In_PosCmd:REAL;
	In_MoveXLock:BOOL;	(*Mechanical Interlock*)
	Out_Ready:BOOL;
	Out_Busy:BOOL;
	Out_InPos:BOOL;
	Out_Referenced:BOOL;
	Out_PosLimit:BOOL;	(*1=OK*)
	Out_NegLimit:BOOL;	(*1=OK*)
	Out_Error:BOOL;
	Out_Warning:BOOL;
	Out_ErrorWord:WORD;
	Out_CurrPos:REAL;
	Out_CurrVel:REAL;
	Out_PosDirc:BOOL;	(*Moving in Positive Direction*)
	Out_NegDirc:BOOL;	(*Moving in Negative Direction*)

END_STRUCT
END_TYPE

// ---- DUTs/structMachineCtrl.TcDUT
TYPE structMachineCtrl :
STRUCT
(* Mode Bit*)
	AutoMode		:BOOL;
	ManualMode		:BOOL;

(* Status Bit*)
	DryRun			:BOOL;
	Stop			:BOOL;
	AutoRunning		:BOOL;
	StopPressed		:BOOL;
	IdleState		:BOOL;
	
	ResetPressed	:BOOL;

	StationStopErr 	:BOOL;
	Warning			:BOOL;
	WarningBuzzer	:BOOL;
	Trouble			:BOOL;
	ErrDetection		:BOOL;

	OriginSchRun		:BOOL;
	InxOrigin			:BOOL;
	AllOrigin			:BOOL;
	AllStationRdy		:BOOL;
	AllStationNoWP 		:BOOL;
	
	E_EmgStop			: BOOL;
	E_LightCurtain		: BOOL;
	E_AirLow 			: BOOL;
	E_SafetyDoorOpen	: BOOL;
	E_Communication		: BOOL;
	E_IncomingPowerPhase: BOOL;
		
	
	
END_STRUCT
END_TYPE

// ---- DUTs/structMachineData.TcDUT
TYPE structMachineData :
STRUCT
	Cnt_TotalGood		:DWORD;
	Cnt_TotalNG			:DWORD;
	Cnt_TotalOutput		:DWORD;
	Cnt_TotalYield		:REAL;
	
	CycleTimeSec		:REAL;	(*Machine cycle time in Seconds*)
	IdleTimeSec			:REAL;	(*Machine idle time in Seconds - waiting for products*)
	CycleTimeSecAvg		:REAL;	(*Machine average cycle time in Seconds*)
	IdleTimeSecAvg		:REAL;	(*Machine average idle time in Seconds - waiting for products*)
	
	TotalRunCycles		:DWORD;	(*Machine Total Autorun Cycles*)
	
	TotalMajorDowntimeHour	:DWORD;	(*Machine down due to trouble*)
	TotalMajorDowntimeMin	:INT;
	TotalMajorDowntimeSec	:INT;

	TotalMinorDowntimeHour	:DWORD;	(*Machine down due to minor error*)
	TotalMinorDowntimeMin	:INT;
	TotalMinorDowntimeSec	:INT;

	TotalRuntimeHour		:DWORD;	(*Machine in normal running state*)
	TotalRuntimeMin			:INT;
	TotalRuntimeSec			:INT;

	TotalIdletimeHour		:DWORD;	(*Machine in normal idle state*)
	TotalIdletimeMin		:INT;
	TotalIdletimeSec		:INT;
	
	Cnt_TotalCntRemoved		:INT;
	CartonPerMinute			:INT;
	BundlePerMinute			:INT;
	
	MTBF				:REAL;
	MTBA				:REAL;

END_STRUCT
END_TYPE

// ---- DUTs/structMotorDirect.TcDUT
TYPE structMotorDirect :
STRUCT
	
	IN_DevName:STRING;

	(* Trigger*)
	T_ManOn:BOOL;
	T_ManOff:BOOL;
	In_AutoON:BOOL;
	In_OrgOn:BOOL;

	In_MoveXLock:BOOL;	(*Mechanical Interlock*)

	E_OnErr:BOOL;
	S_OnSig:BOOL;
	S_Running:BOOL;

END_STRUCT
END_TYPE

// ---- DUTs/structMotorInverter.TcDUT
TYPE structMotorInverter :
STRUCT
	
	IN_DevName:STRING;

	(* Trigger*)
	T_ManOn:BOOL;
	T_ManOff:BOOL;
	In_AutoON:BOOL;
	In_OrgOn:BOOL;
	
	In_SpeedSel:INT;	(*Speed Selection 0-3*)
	In_Dirc:BOOL;		(*Direction Selection*)
	
	In_MoveXLock:BOOL;	(*Mechanical Interlock*)
	
	E_OnErr:BOOL;
	S_InvRdy:BOOL;
	S_Running:BOOL;

END_STRUCT
END_TYPE

// ---- DUTs/structRecipe.TcDUT
TYPE structRecipe :
STRUCT

	rCaseA	:REAL;	(*	Min 200mm Max 640mm	*)
	rCaseB	:REAL;	(*	Min 150mm Max 500mm	*)
	rCaseC	:REAL;	(*	Min 180mm Max 640mm	*)
	
	rBundleW	:REAL;	(*	Min 20mm Max 300mm	*)
	rBundleL	:REAL;	(*	Min 70mm Max 320mm	*)
	rBundleH	:REAL;	(*	Min 15mm Max 150mm	*)
	
	iStackX		:INT;	(*	Stack Count in X Direction	*)
	iStackY		:INT;	(*	Stack Count in Y Direction	*)
	iStackZ		:INT;	(*	Stack Count in Z Direction	*)
			
						(*	Note: All Flap Width must be Case B/2	*)
	
	rWeightTarget	:REAL;	(*	Target Weight for Carton in kg	*)
	rWeightTol		:REAL;	(*	Weight Tolerance for Carton in kg	*)

	sDescription	:STRING; (*Recipe Description *)
	
	rGlue_Distance_Fr_Edge			:REAL;
	rGlue_Length					:REAL;	
	
END_STRUCT
END_TYPE

// ---- DUTs/structStationCtrl.TcDUT
TYPE structStationCtrl :
STRUCT

	AutoRun				:BOOL;
	Running				:BOOL;
	Origin				:BOOL;  (* Station Already Origin *)
	Rdy					:BOOL;	(* Station Ready *)
	NoWP 				:BOOL;
	Bypass				:BOOL;	(* Station Bypass *)

	RunStep				:INT;
	RunReq				:BOOL;	(*Station Start Work Request*)
	Done				:BOOL;	(*Station Work Complete*)
	RunCond				:BOOL;	(* Conditions to Start Auto Sequence*)
	
	Run_NextStepPls		:BOOL;	
	Run_PrevStepPls		:BOOL;
	M_Step				:BOOL;
	M_OneCycle			:BOOL;
	
	T_OriginSearch		:BOOL;	(*Station Origin Run Trigger Button*)
	OriginSchRun		:BOOL;	(*Station in Origin Search Running*)
	OriginRunStep		:INT;
	
	Name				:STRING;
	Status				:STRING;
	StatusInt			:INT;
	CycleTime			:TIME;
	CycleTimeSec		:REAL;	(*Station cycle time in Seconds*)
	IdleTimeSec			:REAL;	(*Station idle time in Seconds*)
	CycleTimeSecAvg		:REAL;	(*Station average cycle time in Seconds*)
	IdleTimeSecAvg		:REAL;	(*Station average idle time in Seconds*)

	MajorFault			:BOOL;	(* Station Major Error, Stop Machine Immediately *)
	MinorFault			:BOOL;	(* Station Minor Error / Fault, Stop after all process done *)
	DeviceFault			:BOOL;	(* Station Device Error*)
	SeqFaultWord		:INT;	(* Sequence Error Word Code	*)
	SeqFaultString		:STRING;	(*Sequence Error String Display*)
	Warning				:BOOL;	(* Station Warning *)

	
END_STRUCT
END_TYPE

// ---- DUTs/structStatistic.TcDUT
TYPE structStatistic :
STRUCT
		RecipeName				:STRING;
		ShiftInformation		:STRING;
		
		RejectLeftTape			:DINT;
		RejectRightTape			:DINT;
		RejectUnderWeight		:DINT;
		RejectOverWeight		:DINT;
		RejectCaseRemoved		:DINT;
		GoodCase				:DINT;
		
		Production_Percentage	:REAL;
		Reject_Percentage		:REAL;
		Net_Efficiency			:REAL;
		OEE						:REAL;
		
		RunTime_Second			:DINT;
		ExternalStop_Second		:DINT;
		InternalStop_Second		:DINT;
		WaitingTime_Second		:DINT;
		
		ServiceStop_Number		:DINT;	
		ServiceStop_Second		:DINT;
		StackerFault_Number		:DINT;
		StackerFault_Second		:DINT;
		XPusherFault_Number		:DINT;
		XPusherFault_Second		:DINT;
		YPusherFault_Number		:DINT;
		YPusherFault_Second		:DINT;
		ErectorFault_Number		:DINT;
		ErectorFault_Second		:DINT;
		ExitFault_Number		:DINT;
		ExitFault_Second		:DINT;
		HorizontalFault_Number	:DINT;
		HorizontalFault_Second	:DINT;
		MajorFault_Number		:DINT;
		MajorFault_Second		:DINT;
		
		
		GlueLeft_Number			:DINT;
		GlueRight_Number		:DINT;		
		TapeLeft_Number			:DINT;
		TapeRight_Number		:DINT;		
		
END_STRUCT
END_TYPE

// ---- DUTs/structVacuum.TcDUT
TYPE structVacuum :
STRUCT
	
	IN_Name:				STRING;
	(*Trigger*)
	T_ManVacuum:			BOOL;
	T_ManPurge:				BOOL;

	(*Mechanical Interlock*)
	In_VacuumX:				BOOL;
	In_PurgeX:				BOOL;
	In_AutoVacuum:			BOOL;
	In_AutoPurge:				BOOL;
	In_OrgVacuum:			BOOL;
	In_OrgPurge:				BOOL;

	E_VacuumErr:			BOOL;
	E_PurgeErr:				BOOL;
	S_Vacuum:				BOOL;
	S_Release:				BOOL;


END_STRUCT
END_TYPE

// ---- GVLs/Device/GVL_Cylinder.TcGVL
VAR_GLOBAL
	
ER_FFlapL_Cyl			:fbCylinderCtrl;	 (* 	1Y1 - ERECTOR FRONT FLAP CLOSING CYL SV (LEFT)	*)
ER_FFlapL_Cyl_Var		:structCylinder;	 (* 	1Y1 - ERECTOR FRONT FLAP CLOSING CYL SV (LEFT)	*)
ER_BFlapL_Cyl			:fbCylinderCtrl;	 (* 	1Y2 - ERECTOR BOTTOM FLAP HOLD SV (LEFT)	*)
ER_BFlapL_Cyl_Var		:structCylinder;	 (* 	1Y2 - ERECTOR BOTTOM FLAP HOLD SV (LEFT)	*)
ER_StpL_Cyl				:fbCylinderCtrl;	 (* 	1Y3 - ERECTOR STOPPER CYL SV (LEFT)	*)
ER_StpL_Cyl_Var			:structCylinder;	 (* 	1Y3 - ERECTOR STOPPER CYL SV (LEFT)	*)
ER_FFlapR_Cyl			:fbCylinderCtrl;	 (* 	1Y4 - ERECTOR FRONT FLAP CLOSING CYL SV (RIGHT)	*)
ER_FFlapR_Cyl_Var		:structCylinder;	 (* 	1Y4 - ERECTOR FRONT FLAP CLOSING CYL SV (RIGHT)	*)
ER_BFlapR_Cyl			:fbCylinderCtrl;	 (* 	1Y5 - ERECTOR BOTTOM FLAP HOLD SV (RIGHT)	*)
ER_BFlapR_Cyl_Var		:structCylinder;	 (* 	1Y5 - ERECTOR BOTTOM FLAP HOLD SV (RIGHT)	*)
ER_StpR_Cyl				:fbCylinderCtrl;	 (* 	1Y6 - ERECTOR STOPPER CYL SV (RIGHT)	*)
ER_StpR_Cyl_Var			:structCylinder;	 (* 	1Y6 - ERECTOR STOPPER CYL SV (RIGHT)	*)
ER_Arm_Cyl				:fbCylinderCtrl;	 (* 	1Y7 - ERECTOR ARM CYL SV	*)
ER_Arm_Cyl_Var			:structCylinder;	 (* 	1Y7 - ERECTOR ARM CYL DOWN SV	*)
ER_ArmTilt_Cyl			:fbCylinderCtrl;	 (* 	1Y8 - ERECTOR ARM TILT CYL SV	*)
ER_ArmTilt_Cyl_Var		:structCylinder;	 (* 	1Y8 - ERECTOR ARM TILT CYL SV	*)
ER_RFlapL_Cyl			:fbCylinderCtrl;	 (* 	3Y1 - ERECTOR REAR FLAP CLOSING CYL SV (LEFT)	*)
ER_RFlapL_Cyl_Var		:structCylinder;	 (* 	3Y1 - ERECTOR REAR FLAP CLOSING CYL SV (LEFT)	*)
ER_RFlapR_Cyl			:fbCylinderCtrl;	 (* 	3Y3 - ERECTOR REAR FLAP CLOSING CYL SV (RIGHT)	*)
ER_RFlapR_Cyl_Var		:structCylinder;	 (* 	3Y3 - ERECTOR REAR FLAP CLOSING CYL SV (RIGHT)	*)
ER_BFlapCloseL_Cyl		:fbCylinderCtrl;	 (* 	1Y1 - ERECTOR BOTTOM FLAP CLOSE SV (LEFT)	*)
ER_BFlapCloseL_Cyl_Var	:structCylinder;	 (* 	1Y1 - ERECTOR BOTTOM FLAP CLOSE SV (LEFT)	*)
ER_BFlapCloseR_Cyl		:fbCylinderCtrl;	 (* 	1Y9 - ERECTOR BOTTOM FLAP CLOSE SV (RIGHT)	*)
ER_BFlapCloseR_Cyl_Var	:structCylinder;	 (* 	1Y9 - ERECTOR BOTTOM FLAP CLOSE SV (RIGHT)	*)
EX_SquarenessCylL_Cyl	:fbCylinderCtrl;	 (* 	1Y11 - SQUARENESS CYLINDER BACKWARD (LEFT)	*)
EX_SquarenessCylL_Var	:structCylinder;	 (* 	1Y11 - SQUARENESS CYLINDER BACKWARD (LEFT)	*)
EX_SquarenessCylR_Cyl	:fbCylinderCtrl;	 (* 	2Y9 - SQUARENESS CYLINDER BACKWARD (RIGHT)	*)
EX_SquarenessCylR_Var	:structCylinder;	 (* 	2Y9 - SQUARENESS CYLINDER BACKWARD (RIGHT)	*)
EX_StpCylL_Cyl			:fbCylinderCtrl;	 (* 	2Y12 - EXIT CYLINDER DOWN (LEFT)	*)
EX_StpCylL_Var			:structCylinder;	 (* 	2Y12 - EXIT CYLINDER DOWN (LEFT)	*)
EX_StpCylR_Cyl			:fbCylinderCtrl;	 (* 	2Y10 - EXIT CYLINDER DOWN (RIGHT)	*)
EX_StpCylR_Var			:structCylinder;	 (* 	2Y10 - EXIT CYLINDER DOWN (RIGHT)	*)



ER_CaseGuideL_Cyl			:fbCylinderCtrl;	 (* 	1Y4 - ERECTOR CASE GUIDE SV (LEFT)	*)
ER_CaseGuideL_Cyl_Var		:structCylinder;	 (* 	1Y4 - ERECTOR CASE GUIDE SV (LEFT)	*)
ER_TFlapClsL_Cyl			:fbCylinderCtrl;	 (* 	1Y6 - ERECTOR TOP FLAP CLOSE SV (LEFT)	*)
ER_TFlapClsL_Cyl_Var		:structCylinder;	 (* 	1Y6 - ERECTOR TOP FLAP CLOSE SV (LEFT)	*)
ER_TFlapOpnL_Cyl			:fbCylinderCtrl;	 (* 	1Y7 - ERECTOR TOP FLAP OPEN SV (LEFT)	*)
ER_TFlapOpnL_Cyl_Var		:structCylinder;	 (* 	1Y6 - ERECTOR TOP FLAP OPEN SV (LEFT)	*)
ER_CaseGuideR_Cyl			:fbCylinderCtrl;	 (* 	1Y4 - ERECTOR CASE GUIDE SV (RIGHT)	*)
ER_CaseGuideR_Cyl_Var		:structCylinder;	 (* 	1Y4 - ERECTOR CASE GUIDE SV (RIGHT)	*)
ER_TFlapClsR_Cyl			:fbCylinderCtrl;	 (* 	2Y6 - ERECTOR TOP FLAP CLOSE SV (RIGHT)	*)
ER_TFlapClsR_Cyl_Var		:structCylinder;	 (* 	1Y6 - ERECTOR TOP FLAP CLOSE SV (RIGHT)	*)
ER_TFlapOpnR_Cyl			:fbCylinderCtrl;	 (* 	1Y6 - ERECTOR TOP FLAP OPEN SV (RIGHT)	*)
ER_TFlapOpnR_Cyl_Var		:structCylinder;	 (* 	1Y6 - ERECTOR TOP FLAP OPEN SV (RIGHT)	*)

ER_NordsonL_Cyl				:fbCylinderCtrl;	 (* 	 ERECTOR NORDSON SV (LEFT)	*)
ER_NordsonL_Cyl_Var			:structCylinder;	 (* 	 ERECTOR NORDSON SV (LEFT)	*)
ER_NordsonR_Cyl				:fbCylinderCtrl;	 (* 	 ERECTOR NORDSON SV (RIGHT)	*)
ER_NordsonR_Cyl_Var			:structCylinder;	 (* 	 ERECTOR NORDSON SV (RIGHT)	*)
				

CO_StkRel_Cyl			:fbCylinderCtrl;	 (* 	2Y2 - COLLATOR STACK RELEASE CYLINDER FWD SV	*)
CO_StkRel_Cyl_Var		:structCylinder;	 (* 	2Y2 - COLLATOR STACK RELEASE CYLINDER FWD SV	*)
CO_Brdg_Cyl				:fbCylinderCtrl;	 (* 	2Y3 - COLLATOR PUSHER BRIDGE CYL SV	*)
CO_Brdg_Cyl_Var			:structCylinder;	 (* 	2Y3 - COLLATOR PUSHER BRIDGE CYL SV	*)
CO_FlapGuide_Cyl		:fbCylinderCtrl;	 (* 	2Y4 - COLLATOR PUSHER GUIDE FLAP CYL SV	*)
CO_FlapGuide_Cyl_Var	:structCylinder;	 (* 	2Y4 - COLLATOR PUSHER GUIDE FLAP CYL SV	*)
(*CO_RFlapGuide_Cyl	:fbCylinderCtrl;	 (* 	2Y3 - COLLATOR PUSHER REAR GUIDE FLAP CYL SV	*)
CO_RFlapGuide_Cyl_Var	:structCylinder;	 (* 	2Y3 - COLLATOR PUSHER REAR GUIDE FLAP CYL SV	*)
CO_FFlapGuide_Cyl	:fbCylinderCtrl;	 (* 	2Y4 - COLLATOR PUSHER FRONT GUIDE FLAP CYL SV	*)
CO_FFlapGuide_Cyl_Var	:structCylinder;	 (* 	2Y4 - COLLATOR PUSHER FRONT GUIDE FLAP CYL SV	*)*)
CO_FFlapBrdg_Cyl		:fbCylinderCtrl;	 (* 	2Y5 - COLLATOR PUSHER FRONT GUIDE FLAP BRIDGE CYL SV	*)
CO_FFlapBrdg_Cyl_Var	:structCylinder;	 (* 	2Y5 - COLLATOR PUSHER FRONT GUIDE FLAP BRIDGE CYL SV	*)
CO_YPush_Strk_Cyl		:fbCylinderCtrl;	 (* 	2Y7 - COLLATOR Y PUSHER STROKE CYL SV	*)
CO_YPush_Strk_Cyl_Var	:structCylinder;	 (* 	2Y7 - COLLATOR Y PUSHER STROKE CYL SV	*)
CO_YPush_Cyl			:fbCylinderCtrl;	 (* 	11Y1 - COLLATOR Y-PUSHER CYL SV	*)
CO_YPush_Cyl_Var		:structCylinder;	 (* 	11Y1 - COLLATOR Y-PUSHER CYL SV	*)
CO_PalletLoc_Cyl		:fbCylinderCtrl;	 (* 	11Y1 - COLLATOR Y-PUSHER CYL SV	*)
CO_PalletLoc_Cyl_Var	:structCylinder;	 (* 	11Y1 - COLLATOR Y-PUSHER CYL SV	*)
CO_Sing1_Cyl			:fbCylinderCtrl;	 (* 	11Y1 - COLLATOR Y-PUSHER CYL SV	*)
CO_Sing1_Cyl_Var		:structCylinder;	 (* 	11Y1 - COLLATOR Y-PUSHER CYL SV	*)
CO_Sing2_Cyl			:fbCylinderCtrl;	 (* 	11Y1 - COLLATOR Y-PUSHER CYL SV	*)
CO_Sing2_Cyl_Var		:structCylinder;	 (* 	11Y1 - COLLATOR Y-PUSHER CYL SV	*)


EL_TapeOpening_Var		:structCylinder;	 (* 	4Y1 - VERTICAL TAPE OPENING CYL FWD SV	*)
EL_TapeOpening_Cyl		:fbCylinderCtrl;	 (* 	4Y1 - VERTICAL TAPE OPENING CYL FWD SV	*)
EL_Tilt_Cyl_Var			:structCylinder;	 (* 	4Y2 - VERTICAL EXIT TILT CYL SV	*)
EL_TiltLift_Cyl			:fbCylinderCtrl;	 (* 	4Y2 - VERTICAL EXIT TILT LIFT CYL SV	*)
EL_EL_TapeLock_Var		:structCylinder;	 (* 	4Y3 - VERTICAL WA TAPE LOCK ACTIVE SV	*)
EL_EL_TapeLock_Cyl		:fbCylinderCtrl;	 (* 	4Y3 - VERTICAL WA TAPE LOCK ACTIVE SV	*)
EL_Tilt_Vac_Lift_Var	:structCylinder;	 (* 	4Y4 - VERTICAL EXIT TILT VAC CYL SV	*)
EL_Tilt_Vac_Lift_Cyl	:fbCylinderCtrl;	 (* 	4Y4 - VERTICAL EXIT TILT VAC CYL SV	*)
EL_TapeChange_Var		:structCylinder;	 (* 	4Y5 - VERTICAL EXIT TILT VAC CYL SV	*)
EL_TapeChange_Cyl		:fbCylinderCtrl;	 (* 	4Y5 - VERTICAL EXIT TILT VAC CYL SV	*)


EL_PushRot_Cyl			:fbCylinderCtrl;	 (* 	5Y1 - ELEVATOR PUSHER ROTATE CYL SV	*)
EL_PushRot_Cyl_Var		:structCylinder;	 (* 	5Y1 - ELEVATOR PUSHER ROTATE CYL SV	*)
EL_Pusher_Cyl			:fbCylinderCtrl;	 (* 	5Y2 - ELEVATOR PUSHER ROTATE CYL SV	*)
EL_Pusher_Cyl_Var		:structCylinder;	 (* 	5Y2 - ELEVATOR PUSHER ROTATE CYL SV	*)







				
EX_FlapHoldL_Cyl		:fbCylinderCtrl_2Station;	 (* 	3Y2 - EXIT FLAP HOLDER LEFT CYL SV (FOR GLUE DISPENSING)	*)
EX_FlapHoldL_Cyl_Var	:structCylinder;	 (* 	3Y2 - EXIT FLAP HOLDER LEFT CYL SV (FOR GLUE DISPENSING)	*)
EX_FlapHoldR_Cyl		:fbCylinderCtrl_2Station;	 (* 	3Y4 - EXIT FLAP HOLDER RIGHT CYL SV (FOR GLUE DISPENSING)	*)
EX_FlapHoldR_Cyl_Var	:structCylinder;	 (* 	3Y4 - EXIT FLAP HOLDER RIGHT CYL SV (FOR GLUE DISPENSING)	*)
EL_TapeL_Cyl			:fbCylinderCtrl;	 (* 	3Y5 - EXIT TAPE EXCHANGE LEFT CYL SV	*)
EL_TapeL_Cyl_Var		:structCylinder;	 (* 	3Y5 - EXIT TAPE EXCHANGE LEFT CYL SV	*)
EL_TapeR_Cyl			:fbCylinderCtrl;	 (* 	3Y6 - EXIT TAPE EXCHANGE RIGHT CYL SV	*)
EL_TapeR_Cyl_Var		:structCylinder;	 (* 	3Y6 - EXIT TAPE EXCHANGE RIGHT CYL SV	*)
EL_Tilt_Cyl				:fbCylinderCtrl;	 (* 	3Y7 - VERTICAL EXIT TILT CYL SV	*)

EL_TiltLift_Cyl_Var	:structCylinder;	 (* 	3Y8 - VERTICAL EXIT TILT LIFT CYL SV	*)

EL_BrakeRel_Cyl	:fbCylinderCtrl;	 (* 	9Y1 - ELEVATOR PUSHER ROTATE CYL SV	*)
EL_BrakeRel_Cyl_Var	:structCylinder;	 (* 	9Y1 - ELEVATOR PUSHER ROTATE CYL SV	*)

EL_FlapHoldL_Cyl	:fbCylinderCtrl;	 (* 	3Y9 - ELEVATOR FLAP HOLDING CYLINDER LEFT SV	*)
EL_FlapHoldL_Cyl_Var	:structCylinder;	  (* 	3Y9 - ELEVATOR FLAP HOLDING CYLINDER LEFT SV	*)
EL_FlapHoldR_Cyl	:fbCylinderCtrl;	 (* 	3Y9 - ELEVATOR FLAP HOLDING CYLINDER RIGHT SV	*)
EL_FlapHoldR_Cyl_Var	:structCylinder;	  (* 	3Y9 - ELEVATOR FLAP HOLDING CYLINDER RIGHT SV	*)

				
EX_90Deg_Cyl		:fbCylinderCtrl;	 (* 	CYL SV FOR 90Deg Conveyor Cylinder	*)
EX_Deg_Cyl_Var		:structCylinder;

END_VAR

// ---- GVLs/Device/GVL_Motor.TcGVL
VAR_GLOBAL
	
ER_VacPump_Mtr		:fbVacuumPumpCtrl;	 (* 	VACUUM PUMP DIRECT ONLINE CONTROL WITH STARTER	*)
ER_VacPump_Mtr_Var	:structMotorDirect;	 (* 	VACUUM PUMP DIRECT ONLINE CONTROL WITH STARTER	*)

ER_BufCvL_Mtr		:fbMotorDirectCtrl;	 (* 	ERECTOR CARTON BUFFER CONVEYOR 	*)
ER_BufCvL_Mtr_Var	:structMotorDirect;	 (* 	ERECTOR CARTON BUFFER CONVEYOR	*)

ER_BufCvR_Mtr		:fbMotorDirectCtrl;	 (* 	ERECTOR CARTON BUFFER CONVEYOR 	*)
ER_BufCvR_Mtr_Var	:structMotorDirect;	 (* 	ERECTOR CARTON BUFFER CONVEYOR	*)

CO_Brake_Clutch		:fbVacuumPumpCtrl;	 (* 	COLLACTOR BRAKE & CLUTCH	*)
CO_Brake_Clutch_Var	:structMotorDirect;	 (* 	COLLACTOR BRAKE & CLUTCH	*)



WT_Mtr	:fbMotorDirectCtrl;	 (* 	WEIGHT CHECKING CONVEYOR 	*)
WT_Mtr_Var	:structMotorDirect;	 (* 	WEIGHT CHECKING CONVEYOR	*)

EL_BotCv_Mtr	:fbMotorDirectCtrl;	 (* 	ELEVATOR BOTTOM EXIT CONVEYOR 	*)
EL_BotCv_Mtr_Var	:structMotorDirect;	 (* 	ELEVATOR BOTTOM EXIT CONVEYOR	*)

EL_TopCv_Mtr	:fbMotorDirectCtrl;	 (* 	ELEVATOR TOP EXIT CONVEYOR 	*)
EL_TopCv_Mtr_Var	:structMotorDirect;	 (* 	ELEVATOR TOP EXIT CONVEYOR	*)

EX_BotCv_Mtr	:fbMotorDirectCtrl;	 (* 	HORIZONTAL BOTTOM EXIT LEFT CONVEYOR  	*)
EX_BotCv_Mtr_Var	:structMotorDirect;	 (* 	HORIZONTAL BOTTOM EXIT LEFT CONVEYOR	*)

EX_TopCv_Mtr	:fbMotorDirectCtrl;	 (* 	HORIZONTAL TOP EXIT LEFT CONVEYOR 	*)
EX_TopCv_Mtr_Var	:structMotorDirect;	 (* 	HORIZONTAL TOP EXIT LEFT CONVEYOR	*)

CO_CV_Mtr	:fbMotorInverterCtrl;	 (* 	COLLATOR INFEED CONVEYOR 	*)
CO_CV_Mtr_Var	:structMotorInverter;	 (* 	COLLATOR INFEED  CONVEYOR	*)

CO_Stk_Mtr	:fbMotorInverterCtrl;	 (* 	COLLATOR STACKING CONVEYOR 	*)
CO_Stk_Mtr_Var	:structMotorInverter;	 (* 	COLLATOR STACKING  CONVEYOR	*)

HOR_BotCv_Mtr	:fbMotorInverterCtrl;	 (* 	HORIZONTAL BOTTOM EXIT CONVEYOR 	*)
HOR_BotCv_Mtr_Var	:structMotorInverter;	 (* 	HORIZONTAL BOTTOM EXIT CONVEYOR	*)

HOR_TopCv_Mtr	:fbMotorInverterCtrl;	 (* 	HORIZONTAL TOP EXIT CONVEYOR 	*)
HOR_TopCv_Mtr_Var	:structMotorInverter;	 (* 	HORIZONTAL TOP EXIT CONVEYOR	*)

HOR_Tilt_In_Mtr	:fbMotorDirectCtrl;	 (* 	Tilt In CONVEYOR 	*)
HOR_Tilt_In_Mtr_Var	:structMotorDirect;	 (* 	Tilt In CONVEYOR	*)

HOR_Tilt_Out_Mtr	:fbMotorDirectCtrl;	 (* 	Tilt Out CONVEYOR 	*)
HOR_Tilt_Out_Mtr_Var	:structMotorDirect;	 (* 	Tilt Out CONVEYOR	*)

CO_UpStreamCv_Mtr		:fbMotorInverterCtrl;	 (* 	COLLATOR UPSTREAM CONVEYOR 	*)
CO_UpStreamCv_Mtr_Var	:structMotorInverter;	 (* 	COLLATOR UPSTREAM  CONVEYOR	*)

END_VAR

// ---- GVLs/Device/GVL_Nordson.TcGVL
VAR_GLOBAL
	ER_Nordson_PumpOnOff_Var			:structMotorDirect;	 (* 	 NORDSON PUMP OFF	*)
	ER_Nordson_Standby_Var				:structMotorDirect;	 (* 	 NORDSON PUMP OFF	*)
	ER_Nordson_HeaterOn_Var				:structMotorDirect;	 (* 	 NORDSON PUMP OFF	*)
	
END_VAR

// ---- GVLs/Device/GVL_Servo.TcGVL
VAR_GLOBAL

	(*ER_M3 Erector Arm Motor - 10M1*)
	ER_Arm_Srv_Input AT %I*:st_Indradrive_DCP_input ;
	ER_Arm_Srv_State AT %I*:UINT ;
	ER_Arm_Srv_Output AT %Q*: st_Indradrive_DCP_output;
	ER_Arm_Srv_Feedrate AT %Q*: UINT;
	ER_Arm_Srv_Drive: fbIndradrive;
	ER_Arm_Srv_Var:structIndradrive;

	(*ER_WA_M5 Erector Width Adjust Motor 1 - 11M1*)
	ER_WA_Srv_Input AT %I*:st_Indradrive_DCP_input ;
	ER_WA_Srv_State AT %I*:UINT ;
	ER_WA_Srv_Output AT %Q*: st_Indradrive_DCP_output;
	ER_WA_Srv_Feedrate AT %Q*: UINT;
	ER_WA_Srv_Drive: fbIndradrive;
	ER_WA_Srv_Var:structIndradrive;

	(*CO_M5 Collator Y Pusher Motor- 111M1*)
	CO_YPush_Srv_Input AT %I*:st_Indradrive_DCP_input ;
	CO_YPush_Srv_State AT %I*:UINT ;
	CO_YPush_Srv_Output AT %Q*: st_Indradrive_DCP_output;
	CO_YPush_Srv_Feedrate AT %Q*: UINT;
	CO_YPush_Srv_Drive: fbIndradrive;
	CO_YPush_Srv_Var:structIndradrive;

	(*EX_WA_M1 Exit Left Height Width Adjust Motor - 12M1*)
	EX_HeightL_WA_Srv_Input AT %I*:st_Indradrive_DCP_input ;
	EX_HeightL_WA_Srv_State AT %I*:UINT ;
	EX_HeightL_WA_Srv_Output AT %Q*: st_Indradrive_DCP_output;
	EX_HeightL_WA_Srv_Feedrate AT %Q*: UINT;
	EX_HeightL_WA_Srv_Drive: fbIndradrive;
	EX_HeightL_WA_Srv_Var:structIndradrive;

	(*EX_WA_M2 Exit Right Height Width Adjust Motor - 13M1*)
	EX_HeightR_WA_Srv_Input AT %I*:st_Indradrive_DCP_input ;
	EX_HeightR_WA_Srv_State AT %I*:UINT ;
	EX_HeightR_WA_Srv_Output AT %Q*: st_Indradrive_DCP_output;
	EX_HeightR_WA_Srv_Feedrate AT %Q*: UINT;
	EX_HeightR_WA_Srv_Drive: fbIndradrive;
	EX_HeightR_WA_Srv_Var:structIndradrive;

	(*EX_WA_M4 Erector Exit Width Adjust Motor - 114M1*)
	EX_WA_Srv_Input AT %I*:st_Indradrive_DCP_input ;
	EX_WA_Srv_State AT %I*:UINT ;
	EX_WA_Srv_Output AT %Q*: st_Indradrive_DCP_output;
	EX_WA_Srv_Feedrate AT %Q*: UINT;
	EX_WA_Srv_Drive: fbIndradrive;
	EX_WA_Srv_Var:structIndradrive;


	(*EX_WA_M3 Exit Left Top Guide Adjust Motor - 124M1*)
	EX_TopL_WA_Srv_Input AT %I*:st_Indradrive_DCP_input ;
	EX_TopL_WA_Srv_State AT %I*:UINT ;
	EX_TopL_WA_Srv_Output AT %Q*: st_Indradrive_DCP_output;
	EX_TopL_WA_Srv_Feedrate AT %Q*: UINT;
	EX_TopL_WA_Srv_Drive: fbIndradrive;
	EX_TopL_WA_Srv_Var:structIndradrive;

	(*EX_WA_M5 Exit Right Top Guide Adjust Motor - 125M1*)
	EX_TopR_WA_Srv_Input AT %I*:st_Indradrive_DCP_input ;
	EX_TopR_WA_Srv_State AT %I*:UINT ;
	EX_TopR_WA_Srv_Output AT %Q*: st_Indradrive_DCP_output;
	EX_TopR_WA_Srv_Feedrate AT %Q*: UINT;
	EX_TopR_WA_Srv_Drive: fbIndradrive;
	EX_TopR_WA_Srv_Var:structIndradrive;


	(*Tilt Servo*)
	EX_Tilt_Srv_Input AT %I*:st_Indradrive_DCP_input ;
	EX_Tilt_Srv_State AT %I*:UINT ;
	EX_Tilt_Srv_Output AT %Q*: st_Indradrive_DCP_output;
	EX_Tilt_Srv_Feedrate AT %Q*: UINT;
	EX_Tilt_Srv_Drive: fbIndradrive;
	EX_Tilt_Srv_Var:structIndradrive;
	
END_VAR

// ---- GVLs/Device/GVL_Vacuum.TcGVL
VAR_GLOBAL
	
ER_BFlapL_Vac	:fbVacuumValveCtrl;	 (* 	4Y1 - ERECTOR LEFT FLAP VACUUM VALVE ON	*)
ER_BFlapL_Vac_Var	:structVacuum;	 (* 	4Y1 - ERECTOR FRONT FLAP CLOSING CYL SV (LEFT)	*)
ER_BFlapR_Vac	:fbVacuumValveCtrl;	 (* 	5Y1 - ERECTOR RIGHT FLAP VACUUM VALVE ON	*)
ER_BFlapR_Vac_Var	:structVacuum;	 (* 	5Y1 - ERECTOR RIGHT FLAP VACUUM VALVE ON	*)
ER_Arm_Vac	:fbVacuumValveCtrl;	 (* 	6Y1 - ERECTOR ARM VACUUM VALVE ON	*)
ER_Arm_Vac_Var	:structVacuum;	 (* 	6Y1 - ERECTOR ARM VACUUM VALVE ON	*)
EL_Tilt_Vac	:fbVacuumValveCtrl;	 (* 	7Y1 - EXIT TILT UNIT VACUUM VALVE ON	*)
EL_Tilt_Vac_Var	:structVacuum;	 (* 	7Y1 - EXIT TILT UNIT VACUUM VALVE ON	*)
EL_Center_Vac	:fbVacuumValveCtrl;	 (* 	10Y1 - ELEVATOR CARTON CENTERING VACUUM ON	*)
EL_Center_Vac_Var	:structVacuum;	 (* 	10Y1 - ELEVATOR CARTON CENTERING VACUUM ON	*)


END_VAR

// ---- GVLs/IO/GVL_Ethercat.TcGVL
VAR_GLOBAL

	S_ECat_NOK:BOOL;
	
	I_ECat_41BC1 	AT %I*	:UINT;
	I_ECat_41DI1 	AT %I*	:UINT;
	I_ECat_41DI2 	AT %I*	:UINT;
	I_ECat_41DO1 	AT %I*	:UINT;
	I_ECat_41DO2 	AT %I*	:UINT;
	I_ECat_41CO1 	AT %I*	:UINT;	
	I_ECat_41BC2 	AT %I*	:UINT;
	I_ECat_41BC3 	AT %I*	:UINT;
	I_ECat_70A1 	AT %I*	:UINT;
	I_ECat_71A1 	AT %I*	:UINT;
	I_ECat_60A1 	AT %I*	:UINT;
	I_ECat_61A1 	AT %I*	:UINT;
	I_ECat_62A1 	AT %I*	:UINT;
	I_ECat_63A1 	AT %I*	:UINT;
	I_ECat_64A1 	AT %I*	:UINT;
	I_ECat_65A1 	AT %I*	:UINT;
	I_ECat_66A1 	AT %I*	:UINT;

	I_ECat_141BC1 	AT %I*	:UINT;
	I_ECat_141DI1 	AT %I*	:UINT;
	I_ECat_141DO1 	AT %I*	:UINT;
	I_ECat_141BC2 	AT %I*	:UINT;
	I_ECat_170A1 	AT %I*	:UINT;
	I_ECat_160A1 	AT %I*	:UINT;
	I_ECat_161A1 	AT %I*	:UINT;
	I_ECat_162A1 	AT %I*	:UINT;
	I_ECat_163A1 	AT %I*	:UINT;
	
	I_ECat_241BC1 	AT %I*	:UINT;
	I_ECat_241DI1 	AT %I*	:UINT;
	I_ECat_241DO1 	AT %I*	:UINT;
	I_ECat_260A1 	AT %I*	:UINT;
	
	I_ECat_341BC1 	AT %I*	:UINT;
	I_ECat_341DI1 	AT %I*	:UINT;
	I_ECat_341DO1 	AT %I*	:UINT;
	I_ECat_341BC2 	AT %I*	:UINT;
	I_ECat_370A1 	AT %I*	:UINT;
	I_ECat_360A1 	AT %I*	:UINT;
	I_ECat_361A1 	AT %I*	:UINT;
	I_ECat_362A1 	AT %I*	:UINT;
	I_ECat_363A1 	AT %I*	:UINT;
	I_ECat_364A1 	AT %I*	:UINT;
	I_ECat_365A1 	AT %I*	:UINT;

END_VAR

// ---- GVLs/IO/GVL_IO_CO.TcGVL
VAR_GLOBAL
	
(**************************************************************************)
(*Collator & Exit Main COntrol Panel*)

IW_141DI1					AT %IB100:WORD;
I_CO_Cv_InvRdy				AT %IX100.0	:BOOL;	 (* 	COLLATOR INFEED CONVEYOR INVERTER READY	*)
I_CO_Stk_InvRdy				AT %IX100.1	:BOOL;	 (* 	COLLATOR STACKING INVERTER READY	*)
IX1002						AT %IX100.2	:BOOL;	 (* 	SPARE	*)
I_Nord_Rdy					AT %IX100.3	:BOOL;	 (* 	NORDSON DISPENSER READY	*)
I_Nord_Alm					AT %IX100.4	:BOOL;	 (* 	NORDSON DISPENSER FAULT	*)
I_Nord_TankLow				AT %IX100.5	:BOOL;	 (* 	NORSON TANK LOW SIGNAL	*)
I_UpStreamInfeedRdy			AT %IX100.6	:BOOL;	 (* 	UPSTREAM INFEED CONVEYOR READY	*)
I_PressSw_OK				AT %IX100.7	:BOOL;	 (* 	INCOMING AIR PRESSURE SWITCH OK	*)

I_Pneumatic_Sup1_ON			AT %IX101.0	:BOOL;	 (* 	Compress Air Supply Coil 1 ON Feedback	*)
I_Pneumatic_Sup2_ON			AT %IX101.1	:BOOL;	 (* 	Compress Air Supply Coil 2 ON feedback	*)
I_COL_Front_Door_Sen		AT %IX101.2	:BOOL;	 (* 	Collator Front Door Sensor	*)
I_COL_Rear_Door_Sen			AT %IX101.3	:BOOL;	 (* 	Collator Rear Door Sensor	*)
IX1014						AT %IX101.4	:BOOL;	 (* 	SPARE	*)
IX1015						AT %IX101.5	:BOOL;	 (* 	SPARE	*)
IX1016						AT %IX101.6	:BOOL;	 (* 	SPARE	*)
IX1017						AT %IX101.7	:BOOL;	 (* 	SPARE	*)

QW_141DO1					AT %QB100:WORD;						    						
O_CO_CV_Mtr_Run				AT %QX100.0	:BOOL;	 (* 	COLLATOR INFEED CONVEYOR INVERTER RUN	*)
O_CO_CV_Mtr_Dirc			AT %QX100.1	:BOOL;	 (* 	COLLATOR INFEED CONVEYOR INVERTER DIRECTION	*)
O_CO_CV_Mtr_Spd1			AT %QX100.2	:BOOL;	 (* 	COLLATOR INFEED CONVEYOR SPEED BIT1	*)
O_CO_CV_Mtr_Spd2			AT %QX100.3	:BOOL;	 (* 	COLLATOR INFEED CONVEYOR SPEED BIT2	*)
O_CO_Stk_Mtr_Run			AT %QX100.4	:BOOL;	 (* 	COLLATOR STACKING INVERTER RUN	*)
O_CO_Stk_Mtr_Dirc			AT %QX100.5	:BOOL;	 (* 	COLLATOR STACKING INVERTER DIRECTION	*)
O_CO_Stk_Mtr_Spd1			AT %QX100.6	:BOOL;	 (* 	COLLATOR STACKING SPEED BIT1	*)
O_CO_Stk_Mtr_Spd2			AT %QX100.7	:BOOL;	 (* 	COLLATOR STACKING SPEED BIT2	*)
						
O_CO_Stk_Mtr_ClutchBrake	AT %QX101.0	:BOOL;	 (* 	COLLATOR STACKING CLUTCH & BRAKE	*)
O_VacPump_On				AT %QX101.1	:BOOL;	 (* 	VACUUM PUMP ON	*)
O_Nord_Auto					AT %QX101.2	:BOOL;	 (* 	NORDSON DISPENSER AUTO STANDBY	*)
O_Nord_Standby				AT %QX101.3	:BOOL;	 (* 	NORDSON DISPENSER STANDBY ON	*)
O_Nord_HeaterOn				AT %QX101.4 :BOOL;	 (* 	NORDSON HEATER ON	*)
O_UpStreamInfeedCv			AT %QX101.5	:BOOL;	 (* 	UPSTREAM INFEED CONVEYOR	*)
QX1016						AT %QX101.6	:BOOL;	 (* 	SAPRE	*)
QX1017						AT %QX101.7	:BOOL;	 (* 	SAPRE	*)

(**************************************************************************)
(*Collactor Field IO - 160A1*)
(*Collator Assembly - Valve Reed Switch*)

IW_160A1					AT %IB110:WORD;
I_CO_YPush_Up	 			AT %IX110.0	:BOOL;	 (* 	COLLATOR X PUSHER CYL UP RS	*)
I_CO_YPush_Dn				AT %IX110.1	:BOOL;	 (* 	COLLATOR X PUSHER CYL DN RS	*)
I_CO_YPush_Strk_Fwd			AT %IX110.2	:BOOL;	 (* 	COLLATOR Y PUSHER STROKE CYL FWD RS	*)
I_CO_YPush_Strk_Bwd			AT %IX110.3	:BOOL;	 (* 	COLLATOR Y PUSHER STROKE CYL BWD RS	*)
I_CO_Brdg_Fwd				AT %IX110.4	:BOOL;	 (* 	COLLATOR PUSHER BRIDGE CYL FWD RS	*)
I_CO_Brdg_Bwd				AT %IX110.5	:BOOL;	 (* 	COLLATOR PUSHER BRIDGE CYL BWD RS	*)
I_CO_FFlapGuide_Fwd			AT %IX110.6	:BOOL;	 (* 	COLLATOR PUSHER FRONT GUIDE FLAP CYL FWD RS	*)
I_CO_FFlapGuide_Bwd			AT %IX110.7	:BOOL;	 (* 	COLLATOR PUSHER FRONT GUIDE FLAP CYL BWD RS	*)


(**************************************************************************)
(*Collactor Field IO - 161A1*)
(*Collator Assembly - Valve Reed Switch & Sensors*)

IW_161A1					AT %IB111:WORD;
I_CO_RFlapGuide_Fwd			AT %IX111.0	:BOOL;	 (* 	COLLATOR PUSHER REAR GUIDE FLAP CYL FWD RS	*)
I_CO_RFlapGuide_Bwd			AT %IX111.1	:BOOL;	 (* 	COLLATOR PUSHER REAR GUIDE FLAP CYL BWD RS	*)
I_CO_PalletInPosition		AT %IX111.2	:BOOL;	 (* 	Pallet In Position	*)
IX1113						AT %IX111.3	:BOOL;	 (* 	SPARE	*)
I_CO_YStk_AtBuf1_PE			AT %IX111.4	:BOOL;	 (* 	STACK PRESENCE AT PUSHER BUFFER AREA 1 SENSOR	*)
I_CO_YStk_AtBuf2_PE			AT %IX111.5	:BOOL;	 (* 	STACK PRESENCE AT PUSHER BUFFER AREA 2 SENSOR	*)
I_CO_Stk_Mtr_HomePos		AT %IX111.6	:BOOL;	 (* 	STACK MOTOR HOME SENSOR	*)
I_CO_Stk_Mtr_UpPos			AT %IX111.7	:BOOL;	 (* 	STACK MOTOR UP POSITION SENSOR	*)
(*
I_CO_CAM_Sensor				AT %IX111.6	:BOOL;	 (* 	STACK MOTOR CAM SENSOR	*)
I_CO_Torque_Limiter			AT %IX111.7	:BOOL;	 (* 	STACK MOTOR TORQUE LIMITER	*)
*)
(**************************************************************************)
(*Collactor Field IO - 162A1*)
(*Collator Assembly - Stacking Module*)

IW_162A1					AT %IB112:WORD;
I_CO_Bdl_PE1				AT %IX112.0	:BOOL;	 (* 	COLLATOR BUNDLE INFEED COUNTING SENSOR 1	*)
I_CO_Bdl_PE2				AT %IX112.1	:BOOL;	 (* 	COLLATOR BUNDLE INFEED COUNTING SENSOR 2	*)
I_CO_Bdl_PE3				AT %IX112.2	:BOOL;	 (* 	COLLATOR BUNDLE INFEED COUNTING SENSOR 3	*)
I_CO_Bdl_PE4				AT %IX112.3	:BOOL;	 (* 	COLLATOR BUNDLE INFEED COUNTING SENSOR 4	*)
I_CO_Bdl_PE5				AT %IX112.4	:BOOL;	 (* 	COLLATOR BUNDLE INFEED COUNTING SENSOR 5	*)
I_CO_Bdl_PE6				AT %IX112.5	:BOOL;	 (* 	COLLATOR BUNDLE INFEED COUNTING SENSOR 6	*)
I_CO_Bdl_PE7				AT %IX112.6	:BOOL;	 (* 	COLLATOR BUNDLE INFEED COUNTING SENSOR 7	*)
I_CO_Bdl_PE8				AT %IX112.7	:BOOL;	 (* 	COLLATOR BUNDLE INFEED COUNTING SENSOR 8	*)

(**************************************************************************)
(*Collactor Field IO - 163A1*)
(*Collator Assembly - Stacking Module*)

IW_163A1					AT %IB113:WORD;
I_CO_Bdl_ZFull_PE			AT %IX113.0	:BOOL;	 (* 	COLLATOR BUNDLE Z-AXIS STACK FULL SENSOR	*)
I_CO_Bdl_ZLimit_PE			AT %IX113.1	:BOOL;	 (* 	COLLATOR BUNDLE Z-AXIS STACK LIMIT (OVERFLOW) SENSOR	*)
I_CO_Bdl_Stack_PE			AT %IX113.2	:BOOL;	 (* 	COLLATOR BUNDLE AT STACKED UP SENSOR	*)
I_CO_Bdl_DoorSwitch			AT %IX113.3	:BOOL;	 (* 	COLLATOR BUNDLE DOOR SWITCH	*)
I_Upstream_Jam_Sen			AT %IX113.4	:BOOL;	 (* 	COLLATOR UPSTREAM JAM SENSOR *)
IX1135						AT %IX113.5	:BOOL;	 (* 	SPARE	*)
IX1136						AT %IX113.6	:BOOL;	 (* 	SPARE	*)
IX1137						AT %IX113.7	:BOOL;	 (* 	SPARE	*)

(**************************************************************************)
(*Collactor Field IO - 164A1*)
(*Collator Assembly - Stacking Module*)

IW_164A1					AT %IB114:WORD;
I_CO_PTC_PE1				AT %IX114.0	:BOOL;	 (* 	COLLATOR BUNDLE PART CONFIRMATION SENSOR1	*)
I_CO_PTC_PE2				AT %IX114.1	:BOOL;	 (* 	COLLATOR BUNDLE PART CONFIRMATION SENSOR2	*)
I_CO_PTC_PE3				AT %IX114.2	:BOOL;	 (* 	COLLATOR BUNDLE PART CONFIRMATION SENSOR3	*)
I_CO_PTC_PE4				AT %IX114.3	:BOOL;	 (* 	COLLATOR BUNDLE PART CONFIRMATION SENSOR4	*)
I_CO_PTC_PE5				AT %IX114.4	:BOOL;	 (* 	COLLATOR BUNDLE PART CONFIRMATION SENSOR5	*)
I_CO_PTC_PE6				AT %IX114.5	:BOOL;	 (* 	COLLATOR BUNDLE PART CONFIRMATION SENSOR6	*)
I_CO_PTC_PE7				AT %IX114.6	:BOOL;	 (* 	COLLATOR BUNDLE PART CONFIRMATION SENSOR7	*)
I_CO_PTC_PE8				AT %IX114.7	:BOOL;	 (* 	COLLATOR BUNDLE PART CONFIRMATION SENSOR8	*)






I_CO_FxStp_Up				AT %IX110.0	:BOOL;	 (* 	COLLATOR FIXED RAIL CV STOPPER CYL UP RS	*)
I_CO_FxStp_Dn				AT %IX110.1	:BOOL;	 (* 	COLLATOR FIXED RAIL CV STOPPER CYL DN RS	*)


I_CO_Bdl_StackRel_PE		AT %IX110.5	:BOOL;	 (* 	COLLATOR BUNDLE AT STACK RELEASE POSITION SENSOR	*)
I_CO_FxStkRel_Fwd			AT %IX110.6	:BOOL;	 (*		COLLATOR FIXED RAIL STACK RELEASE CYLINDER FWD RS*)
I_CO_FxStkRel_Bwd			AT %IX110.7	:BOOL;	 (*		COLLATOR FIXED RAIL STACK RELEASE CYLINDER BWD RS*) 










O_EL_BotCV_Mtr_On			AT %QX901.1	:BOOL;	 (* 	ELEVATOR BOTTOM EXIT CV STARTER ON	*)
O_EL_TopCV_Mtr_On			AT %QX901.2	:BOOL;	 (* 	ELEVATOR TOP EXIT CV STARTER ON	*)
O_EX_BotCV_Mtr_On			AT %QX901.3	:BOOL;	 (* 	HORIZONTAL BOTTOM EXIT CV 1 STARTER ON	*)
O_EX_TopCV_Mtr_On			AT %QX901.4	:BOOL;	 (* 	HORIZONTAL TOP EXIT CV 2 STARTER ON	*)





IX1005		AT %IX100.5	:BOOL;	 (* 	SPARE	*)

						

I_EL_FlapHoldR_Fwd		AT %IX101.2	:BOOL;	 (* 	ELEVATOR FLAP HOLDING CYLINDER RIGHT FWD RS	*)
I_EL_FlapHoldR_Bwd		AT %IX101.3	:BOOL;	 (* 	ELEVATOR FLAP HOLDING CYLINDER RIGHT BWD RS	*)
I_EL_FlapHoldL_Fwd		AT %IX101.4	:BOOL;	 (* 	ELEVATOR FLAP HOLDING CYLINDER LEFT FWD RS	*)
I_EL_FlapHoldL_Bwd		AT %IX101.5	:BOOL;	 (* 	ELEVATOR FLAP HOLDING CYLINDER LEFT BWD RS	*)










I_CO_MvStp_Up		AT %IX111.0	:BOOL;	 (* 	COLLATOR MOVING RAIL CV STOPPER CYL UP RS	*)
I_CO_MvStp_Dn		AT %IX111.1	:BOOL;	 (* 	COLLATOR MOVING RAIL CV STOPPER CYL DN RS	*)

IX1114		AT %IX111.4	:BOOL;	 (* 	SPARE	*)
I_CO_Bdl_Count_PE2		AT %IX111.5	:BOOL;	 (* 	SPARE	*)
I_CO_MvStkRel_Fwd				AT %IX111.6	:BOOL;	 (*		COLLATOR MOVING RAIL STACK RELEASE CYLINDER FWD RS*)
I_CO_MvStkRel_Bwd				AT %IX111.7	:BOOL;	 (*		COLLATOR MOVING RAIL STACK RELEASE CYLINDER BWD RS*) 






I_CO_Stk_UpPos		AT %IX112.4	:BOOL;	 (* 	COLLATOR STACKING CAM MODULE AT UP POSITION	*)
I_CO_Stk_DnPos		AT %IX112.5	:BOOL;	 (* 	COLLATOR STACKING CAM MODULE AT DOWN POSITION	*)
IX1126		AT %IX112.6	:BOOL;	 (* 	SPARE	*)
IX1127		AT %IX112.7	:BOOL;	 (* 	SPARE	*)




(**************************************************************************)
(*Erector Field IO - 165A1*)
(*Exit Assembly - WEIGHT CHECK & TILT UNIT*)

IW_165A1				AT %IB115:WORD;


I_EL_TiltLift_Fwd		AT %IX115.3	:BOOL;	 (* 	VERTICAL EXIT TILT LIFT CYL FWD RS	*)
I_EL_TiltLift_Bwd		AT %IX115.4	:BOOL;	 (* 	VERTICAL EXIT TILT LIFT CYL BWD RS	*)

IX1156		AT %IX115.6	:BOOL;	 (* 	SPARE	*)
IX1157		AT %IX115.7	:BOOL;	 (* 	SPARE	*)

(**************************************************************************)
(*Erector Field IO - 166A1*)
(*Exit Assembly - ELEVATOR MODULE*)



IX1164		AT %IX116.4	:BOOL;	 (* 	SPARE	*)
IX1165		AT %IX116.5	:BOOL;	 (* 	SPARE	*)
IX1166		AT %IX116.6	:BOOL;	 (* 	SPARE	*)
IX1167		AT %IX116.7	:BOOL;	 (* 	SPARE	*)


(**************************************************************************)
(*Erector Field IO - 167A1*)
(*Exit Assembly - ELEVATOR MODULE*)

QW_167A1				AT %QB110:WORD;



QX1104		AT %QX110.4	:BOOL;	 (* 	SPARE	*)
QX1105		AT %QX110.5	:BOOL;	 (* 	SPARE	*)
QX1106		AT %QX110.6	:BOOL;	 (* 	SPARE	*)
QX1107		AT %QX110.7	:BOOL;	 (* 	SPARE	*)

(**************************************************************************)
(*Erector Field IO - 168A1*)
(*Collator Assembly - Pusher Bridge & Rear Flap Guide*)

IW_168A1				AT %IB117:WORD;



IX1176		AT %IX117.6	:BOOL;	 (* 	SPARE	*)
IX1177		AT %IX117.7	:BOOL;	 (* 	SPARE	*)

(**************************************************************************)
(*Erector Field IO - 169A1*)
(*Collator Assembly - Pusher Bridge & Rear Flap Guide*)

IW_169A1				AT %IB118:WORD;

I_CO_FFlapBrdg_Fwd		AT %IX118.2	:BOOL;	 (* 	COLLATOR PUSHER FRONT GUIDE FLAP BRIDGE CYL FWD RS	*)
I_CO_FFlapBrdg_Bwd		AT %IX118.3	:BOOL;	 (* 	COLLATOR PUSHER FRONT GUIDE FLAP BRIDGE CYL BWD RS	*)

I_CO_Bdl_XFull_PE		AT %IX118.6	:BOOL;	 (* 	COLLATOR BUNDLE X-AXIS STACK FULL SENSOR	*)
I_CO_Bdl_XLimit_PE		AT %IX118.7	:BOOL;	 (* 	COLLATOR BUNDLE X-AXIS STACK LIMIT (OVERFLOW) SENSOR	*)

I_CO_YPush_Gap_PE :BOOL;	(*spare for gap sensor*)



QW119				AT %IB119:WORD;
QX1190				AT %IX119.0	:BOOL;	 

(**************************************************************************)
(*Additional*)
IW_170A1				AT %IB411 : BYTE;
IW_170A2				AT %IB412 : BYTE;	

I_CO_Sing1_Fwd			AT %IX412.0 :BOOL;
I_CO_Sing1_Bwd			AT %IX412.1 :BOOL;
I_CO_Sing2_Fwd			AT %IX412.2 :BOOL;
I_CO_Sing2_Bwd			AT %IX412.3 :BOOL;
I_CO_PalletLocating_Fwd	AT %IX412.4 :BOOL;
I_CO_PalletLocating_Bwd	AT %IX412.5 :BOOL;








END_VAR

// ---- GVLs/IO/GVL_IO_EL.TcGVL
VAR_GLOBAL
(*
(**************************************************************************)
(*VerticalL IO *)

IW_341DI1					AT %IB300:WORD;						    
I_EX_BotCV_Ctn_PE			AT %IX300.0	:BOOL;	 (* 	ERECTOR CARTON PRESENCE AT  BOTTOM EXIT CV. SENSOR SHOULD BE OFF FOR ELEVATOR TO MOVE.	*)
I_EX_TopCV_Ctn_PE			AT %IX300.1	:BOOL;	 (* 	ERECTOR CARTON PRESENCE AT  TOP EXIT CV. SENSOR SHOULD BE OFF FOR ELEVATOR TO MOVE.	*)
I_LC_SC_OK					AT %IX300.2	:BOOL;	 (* 	VERTICAL EXIT LIGHT CURTAIN OK	*)
IX3003						AT %IX300.3	:BOOL;	 (* 	SPARE	*)
IX3004						AT %IX300.4	:BOOL;	 (* 	SPARE	*)
IX3005						AT %IX300.5	:BOOL;	 (* 	SPARE	*)
IX3006						AT %IX300.6	:BOOL;	 (* 	SPARE	*)
IX3007						AT %IX300.7	:BOOL;	 (* 	SPARE	*)

IX3010						AT %IX301.2	:BOOL;	 (* 	SPARE	*)
IX3011						AT %IX301.3	:BOOL;	 (* 	SPARE	*)
IX3012						AT %IX301.2	:BOOL;	 (* 	SPARE	*)
IX3013						AT %IX301.3	:BOOL;	 (* 	SPARE	*)
IX3014						AT %IX301.4	:BOOL;	 (* 	SPARE	*)
IX3015						AT %IX301.5	:BOOL;	 (* 	SPARE	*)
IX3016						AT %IX301.6	:BOOL;	 (* 	SPARE	*)
IX3017						AT %IX301.7	:BOOL;	 (* 	SPARE	*)


(**************************************************************************)
(*VerticalL Field IO *)
IW_360A1					AT %IB310:WORD;
I_EL_Tape_OpeningL_FWD		AT %IX310.0	:BOOL;	 (* 	TAPE OPENING LEFT FWD SENSOR	*)
I_EL_Tape_OpeningL_BWD		AT %IX310.1	:BOOL;	 (* 	TAPE OPENING LEFT BWD SENSOR	*)
I_EL_Tape_OpeningR_FWD		AT %IX310.2	:BOOL;	 (* 	TAPE OPENING RIGHT FWD SENSOR	*)
I_EL_Tape_OpeningR_BWD		AT %IX310.3	:BOOL;	 (* 	TAPE OPENING RIGHT BWD SENSOR	*)
I_EL_Tilt_Fwd				AT %IX310.4	:BOOL;	 (* 	VERTICAL EXIT TILT CYL FWD RS	*)
I_EL_Tilt_Bwd				AT %IX310.5	:BOOL;	 (* 	VERTICAL EXIT TILT CYL BWD RS	*)
I_EL_BeltTensionR_OK		AT %IX310.6	:BOOL;	 (* 	ELEVATOR BELT TENSION RIGHT OK	*)
I_EL_BeltTensionL_OK		AT %IX310.7	:BOOL;	 (* 	ELEVATOR BELT TENSION LEFT OK	*)

IW_361A1					AT %IB311:WORD;
I_EL_Tape_Change_FWD		AT %IX311.0	:BOOL;	 (* 	TAPE CHANGE FWD SENSOR	*)
I_EL_Tape_Change_BWD		AT %IX311.1	:BOOL;	 (* 	TAPE CHANGE BWD SENSOR	*)
I_EL_LOW_EXIT_FULL			AT %IX311.2	:BOOL;	 (* 	ELEVATOR LOW EXIT FULL SENSOR	*)
IX3113						AT %IX311.3	:BOOL;	 (* 	SPARE	*)
IX3114						AT %IX311.4	:BOOL;	 (* 	SPARE	*)
IX3115						AT %IX311.5	:BOOL;	 (* 	SPARE	*)
IX3116						AT %IX311.6	:BOOL;	 (* 	SPARE	*)
IX3117						AT %IX311.7	:BOOL;	 (* 	SPARE	*)

IW_362A1					AT %IB312:WORD;
I_EL_TapeL_Refill_PE		AT %IX312.0	:BOOL;	 (* 	EXIT TAPE LEFT REFILL SENSOR (0=NEED REFILL)	*)
I_EL_TapeL_Empty_PE			AT %IX312.1	:BOOL;	 (* 	EXIT TAPE LEFT EMPTY SENSOR 	*)
I_EL_TapeL_Break_PE			AT %IX312.2	:BOOL;	 (* 	EXIT TAPE LEFT BREAK SENSOR 	*)
I_EL_TapeR_RefilR_PE		AT %IX312.3	:BOOL;	 (* 	EXIT TAPE RIGHT REFILL SENSOR (0=NEED REFILL)	*)
I_EL_TapeR_Empty_PE			AT %IX312.4	:BOOL;	 (* 	EXIT TAPE LEFT EMPTY SENSOR 	*)
I_EL_TapeR_Break_PE			AT %IX312.5	:BOOL;	 (* 	EXIT TAPE LEFT BREAK SENSOR 	*)
I_EL_DriveBeltTension_OK	AT %IX312.6	:BOOL;	 (* 	ELEVATOR DRIVE BELT TENSION OK	*)
I_EL_Tilt_VacSw				AT %IX312.7	:BOOL;	 (* 	VERTICAL EXIT TILT VACUUM SWITCH	*)


QW_341DO1					AT %QB300:WORD;						    
QX3000						AT %QX300.0	:BOOL;	 (* 	SPARE	*)
QX3001						AT %QX300.1	:BOOL;	 (* 	SPARE	*)
QX3002						AT %QX300.2	:BOOL;	 (* 	SPARE	*)
O_EL_LC_Mute1				AT %QX310.3	:BOOL;	 (* 	ELEVATOR - MUTE LIGHT CURTAIN	*)
O_EL_LC_Mute2				AT %QX310.4	:BOOL;	 (* 	ELEVATOR - MUTE LIGHT CURTAIN	*)
QX3005						AT %QX300.5	:BOOL;	 (* 	SPARE	*)
QX3006						AT %QX300.6	:BOOL;	 (* 	SPARE	*)
QX3007						AT %QX300.7	:BOOL;	 (* 	SPARE	*)					


QW_363A1					AT %QB310:WORD;	
O_EL_Tilt_Vac_On			AT %QX310.0	:BOOL;	 (* 	7Y1 - EXIT TILT UNIT VACUUM VALVE ON	*)
QX3101						AT %QX310.3	:BOOL;	 (* 	SPARE	*)
QX3102						AT %QX310.4	:BOOL;	 (* 	SPARE	*)
QX3103						AT %QX310.3	:BOOL;	 (* 	SPARE	*)
QX3104						AT %QX310.4	:BOOL;	 (* 	SPARE	*)
QX3105						AT %QX310.5	:BOOL;	 (* 	SPARE	*)
QX3106						AT %QX310.6	:BOOL;	 (* 	SPARE	*)
QX3107						AT %QX310.7	:BOOL;	 (* 	SPARE	*)

IW_364A1					AT %IB313:WORD;
I_EL_PushRot_Up				AT %IX313.0	:BOOL;	 (* 	ELEVATOR PUSHER ROTATE CYL UP RS	*)
I_EL_PushRot_Dn				AT %IX313.1	:BOOL;	 (* 	ELEVATOR PUSHER ROTATE CYL DN RS	*)
I_EL_Pusher_Fwd				AT %IX313.2	:BOOL;	 (* 	8Y1 - ELEVATOR PUSHER CYL FWD SV	*)
I_EL_Pusher_Bwd				AT %IX313.3	:BOOL;	 (* 	8Y1 - ELEVATOR PUSHER CYL BWD SV	*)
I_EL_Center_VacSw			AT %IX313.4	:BOOL;	 (* 	ELEVATOR CARTON CENTERING VACUUM SWITCH	*)
I_EL_Ctn_PE	 				AT %IX313.5	:BOOL;	 (* 	ELEVATOR PRODUCT PRESENCE ON CV SENSOR	*)
IX3136						AT %IX313.6	:BOOL;	 (* 	SPARE	*)
IX3137						AT %IX313.7	:BOOL;	 (* 	SPARE	*)

QW_365A1					AT %QB311:WORD;	
O_EL_PushRot_Up				AT %QX311.0	:BOOL;	 (* 	8Y1 - ELEVATOR PUSHER ROTATE CYL UP SV	*)
O_EL_PushRot_Dn				AT %QX311.1	:BOOL;	 (* 	8Y1 - ELEVATOR PUSHER ROTATE CYL DN SV	*)
Q_EL_Pusher_Fwd				AT %QX311.2	:BOOL;	 (* 	8Y1 - ELEVATOR PUSHER CYL FWD SV	*)
Q_EL_Pusher_Bwd				AT %QX311.3	:BOOL;	 (* 	8Y1 - ELEVATOR PUSHER CYL BWD SV	*)
O_EL_SafeLock_Rel			AT %QX311.4	:BOOL;	 (* 	9Y1 - ELEVATOR SAFETY LOCK RELEASE SV	*)
O_EL_Center_Vac_On			AT %QX311.5	:BOOL;	 (* 	10Y1 - ELEVATOR CARTON CENTERING VACUUM ON	*)
QX3116						AT %QX311.6	:BOOL;	 (* 	SPARE	*)
QX3117						AT %QX311.7	:BOOL;	 (* 	SPARE	*)
*)
END_VAR

// ---- GVLs/IO/GVL_IO_HOR.TcGVL
VAR_GLOBAL
(**************************************************************************)
(*Horizontal IO *)

IW_241DI1					AT %IB200:WORD;						    
I_HOR_TopCv_InvRdy			AT %IX200.0	:BOOL;	 (* 	HORIZONTAL TOP CONVEYOR INVERTER READY	*)
I_HOR_BotCv_InvRdy			AT %IX200.1	:BOOL;	 (* 	HORIZONTAL BOTTOM CONVEYOR INVERTER READY	*)
I_HLC_SC_OK					AT %IX200.2	:BOOL;	 (* 	HORIZONTAL EXIT LIGHT CURTAIN OK	*)
I_EStop_HorL				AT %IX200.3	:BOOL;	 (* 	EMERGENCY STOP FOR HORIZONTAL LEFT	*)
I_EStop_HorR				AT %IX200.4	:BOOL;	 (* 	EMRGENCT STOP FOR HORIZONTAL RIGHT	*)
I_EStop_HorExit				AT %IX200.5	:BOOL;	 (* 	EMERGENCY STOP FOR HORZONTAL EXIT	*)
I_CO_PusherReady			AT %IX200.6	:BOOL;	 (* 	PUSHER READY	*)
I_EStop_Collator			AT %IX200.7	:BOOL;	 (* 	EMERGENCY STOP FOR COLLATOR	*)

IX2010						AT %IX201.2	:BOOL;	 (* 	SPARE	*)
IX2011						AT %IX201.3	:BOOL;	 (* 	SPARE	*)
IX2012						AT %IX201.2	:BOOL;	 (* 	SPARE	*)
IX2013						AT %IX201.3	:BOOL;	 (* 	SPARE	*)
IX2014						AT %IX201.4	:BOOL;	 (* 	SPARE	*)
IX2015						AT %IX201.5	:BOOL;	 (* 	SPARE	*)
IX2016						AT %IX201.6	:BOOL;	 (* 	SPARE	*)
IX2017						AT %IX201.7	:BOOL;	 (* 	SPARE	*)


(**************************************************************************)
(*Horizontal Field IO *)
IW_260A1					AT %IB210:WORD;
I_HOR_Entry_Cv_Present		AT %IX210.0	:BOOL;	 (* 	HORIZONTAL PRODUCT PRESENCE AT ENTRY CONVEYOR SENSOR	*)
I_HOR_TapeL_Present_PE		AT %IX210.1	:BOOL;	 (* 	HORIZONTAL TAPE LEFT PRESENT SENSOR	*)
I_HOR_TapeR_Present_PE		AT %IX210.2	:BOOL;	 (* 	HORIZONTAL TAPE RIGHT PRESENT SENSOR	*)
I_HOR_DnStream_Cv_Full		AT %IX210.3	:BOOL;	 (* 	HORIZONTAL EXIT CONVEYOR FULL SENSOR	*)
I_HOR_Left_Door				AT %IX210.4	:BOOL;	 (* 	HORIZONTAL EXIT LEFT DOOR SENSOR	*)
I_HOR_Right_Door			AT %IX210.5	:BOOL;	 (* 	HORIZONTAL EXIT RIGHT DOOR SENSOR	*)
I_HOR_TapeL_Empty_PE		AT %IX210.6	:BOOL;	 (* 	HORIZONTAL TAPE LEFT EMPTY SENSOR	*)
I_HOR_TapeR_Empty_PE		AT %IX210.7	:BOOL;	 (* 	HORIZONTAL TAPE RIGHT EMPTY SENSOR	*)

(**************************************************************************)
(*Horizontal Field IO *)
IW_261A1					AT %IB211:WORD;
I_HOR_Tilt_In_Cv_Present	AT %IX211.0	:BOOL;	 (* 	HORIZONTAL TILT CONVEYOR IN SENSOR	*)
I_HOR_Tilt_Out_Cv_present	AT %IX211.1	:BOOL;	 (* 	HORIZONTAL TILT CONVEYOR OUT SENSOR	*)
I_HOR_TiltDoor				AT %IX211.2	:BOOL;	 (* 	HORIZONTAL TILT UNIT DOOR SENSOR	*)


QW_241DO1					AT %QB200:WORD;						    
QX2000						AT %QX200.0	:BOOL;	 (* 	SPARE	*)
O_HOR_LC_Mute1				AT %QX200.1	:BOOL;	 (* 	ELEVATOR - MUTE 1 LIGHT CURTAIN	*)
O_HOR_LC_Mute2				AT %QX200.2	:BOOL;	 (* 	ELEVATOR - MUTE 2 LIGHT CURTAIN	*)
O_HOR_TiltCV1_On			AT %QX200.3	:BOOL;	 (* 	Tilt Conveyer 1	*)
O_HOR_TiltCV2_On			AT %QX200.4	:BOOL;	 (* 	Tilt Conveyer 2	*)
QX2005						AT %QX200.5	:BOOL;	 (* 	SPARE	*)
QX2006						AT %QX200.6	:BOOL;	 (* 	SPARE	*)
QX2007						AT %QX200.7	:BOOL;	 (* 	SPARE	*)					

O_HOR_TopCv_Mtr_Run			AT %QX201.0	:BOOL;	 (* 	HORIZONTAL TOP CONVEYOR INVERTER RUN	*)
O_HOR_TopCv_Mtr_Dirc		AT %QX201.1	:BOOL;	 (* 	HORIZONTAL TOP CONVEYOR INVERTER DIRECTION	*)
O_HOR_TopCv_Mtr_Spd1		AT %QX201.2	:BOOL;	 (* 	HORIZONTAL TOP CONVEYOR SPEED BIT1	*)
O_HOR_TopCv_Mtr_Spd2		AT %QX201.3	:BOOL;	 (* 	HORIZONTAL TOP CONVEYOR SPEED BIT2	*)
O_HOR_BotCv_Mtr_Run			AT %QX201.4	:BOOL;	 (* 	HORIZONTAL BOTTOM CONVEYOR INVERTER RUN	*)
O_HOR_BotCv_Mtr_Dirc		AT %QX201.5	:BOOL;	 (* 	HORIZONTAL BOTTOM CONVEYOR INVERTER DIRECTION	*)
O_HOR_BotCv_Mtr_Spd1		AT %QX201.6	:BOOL;	 (* 	HORIZONTAL BOTTOM CONVEYOR SPEED BIT1	*)
O_HOR_BotCv_Mtr_Spd2		AT %QX201.7	:BOOL;	 (* 	HORIZONTAL BOTTOM CONVEYOR SPEED BIT2	*)


I_HOR_90Deg_Tilt_Cly_Up		AT %IX211.0	:BOOL;	(*		HORIZONTAL 90 Deg TILT CYLINDER UP SENSOR *)
I_HOR_90Deg_Tilt_Cly_Dn		AT %IX211.1	:BOOL;	(*		HORIZONTAL 90 Deg TILT CYLINDER DOWN SENSOR *)
I_HOR_90Deg_Full_PE			AT %IX211.2	:BOOL;	(*		HORIZONTAL 90 Deg TILT FULL SENSOR	*)

O_HOR_90Deg_Cyl_Up			AT	%QX211.0 :BOOL;	(*		HORIZONTAL	90 Deg TILT CYLINDER UP	*)
O_HOR_90Deg_Cyl_Dn			AT	%QX211.1 :BOOL;	(*		HORIZONTAL	90 Deg TILT CYLINDER DOWN	*)

END_VAR

// ---- GVLs/IO/GVL_IO_ER.TcGVL
                                                                                                                                                                                                                                                                                                                                                                                                                                                                                                                                                                                                                                                                                                                                                                                                                                                                                                                                                                                                                                                                                                                                                                                                                                                                                                                                                                                                                                                                                                                                                                                               VAR_GLOBAL

(**************************************************************************)
(*Erector Main COntrol Panel*)

IW_41DI1					AT %IB0:WORD;
I_Start_PB 					AT %IX0.0	:BOOL;	 (* 	START PB	*)
I_Stop_PB					AT %IX0.1	:BOOL;	 (* 	STOP PB	*)
I_Reset_PB					AT %IX0.2	:BOOL;	 (* 	RESET PB	*)
I_Safety_OK					AT %IX0.3	:BOOL;	 (* 	OVERALL SAFETY OK	*)
I_Emg_SC_OK					AT %IX0.4	:BOOL;	 (* 	EMERGENCY OK	*)
I_Door_SC_OK				AT %IX0.5	:BOOL;	 (* 	DOOR SWITCH OK	*)
I_Case_Infeed_Safety_Ok		AT %IX0.6	:BOOL;	 (* 	CASE INFEED SAFETY OK	*)
I_PCUPS_OK					AT %IX0.7	:BOOL;	 (* 	PC UPS OK	*)
					
I_CartonCV_M1M2_OK			AT %IX1.0	:BOOL;	 (* 	CARTON CONVEYOR MOTOR 1&2 STARTER OK	*)
I_Weighing_CV_OK			AT %IX1.1	:BOOL;	 (* 	WEIGHING CONVEYOR STARTER OK	*)
I_IncomingPowerPhase_OK		AT %IX1.2	:BOOL;	 (* 	Incoming Power Phase OK	*)
I_Erector_Front_Door_Sen	AT %IX1.3	:BOOL;	 (* 	Erector Front Door Sensor	*)
I_erector_Rear_Door_Sen		AT %IX1.4	:BOOL;	 (* 	Erector Rear Door Sensor	*)
IX15						AT %IX1.5	:BOOL;	 (* 	SPARE	*)
IX16						AT %IX1.6	:BOOL;	 (* 	SPARE	*)
IX17						AT %IX1.7	:BOOL;	 (* 	SPARE	*)

IW_41DI2					AT %IB2:WORD;						
I_UpStream_ExitJam			AT %IX2.0	:BOOL;	 (* 	UPSTREAM EXIT JAM	*)
I_UpStream_InProd			AT %IX2.1	:BOOL;	 (* 	UPSTREAM IN PRODUCTION	*)
IX22						AT %IX2.2	:BOOL;	 (* 	SPARE	*)
IX23						AT %IX2.3	:BOOL;	 (* 	SPARE	*)
I_DnStream_ExitJam			AT %IX2.4	:BOOL;	 (* 	DOWNSTREAM EXIT JAM	*)
I_DnStream_InProd			AT %IX2.5	:BOOL;	 (* 	DOWNSTREAM IN PRODUCTION	*)
IX26						AT %IX2.6	:BOOL;	 (* 	SPARE	*)
IX27						AT %IX2.7	:BOOL;	 (* 	SPARE	*)
						
I_TnT_Healthy				AT %IX3.0	:BOOL;	 (* 	Track and Trace Healthy	*)
I_TnT_LabelerINP			AT %IX3.1	:BOOL;	 (* 	Track and Trace Labeller In Position	*)
IX32						AT %IX3.2	:BOOL;	 (* 	SPARE	*)
IX33						AT %IX3.3	:BOOL;	 (* 	SPARE	*)
IX34						AT %IX3.4	:BOOL;	 (* 	SPARE	*)
IX35						AT %IX3.5	:BOOL;	 (* 	SPARE	*)
IX36						AT %IX3.6	:BOOL;	 (* 	SPARE	*)
I_EStop_Panel				AT %IX3.7	:BOOL;	 (* 	PANEL EMERGENCY STOP	*)

QW_41DO1					AT %QB0:WORD;						
O_Start_PL					AT %QX0.0	:BOOL;	 (* 	START PB LIGHT	*)
O_Stop_PL					AT %QX0.1	:BOOL;	 (* 	STOP PB LIGHT	*)
O_Reset_PL					AT %QX0.2	:BOOL;	 (* 	RESET PB LIGHT	*)
O_Red_TL					AT %QX0.3	:BOOL;	 (* 	RED TOWER LIGHT	*)
O_Yel_TL					AT %QX0.4	:BOOL;	 (* 	YELLOW TOWER LIGHT	*)
O_Grn_TL					AT %QX0.5	:BOOL;	 (* 	GREEN TOWER LIGHT	*)
O_Buz_TL					AT %QX0.6	:BOOL;	 (* 	BUZZER TOWER LIGHT	*)
O_DoorLock					AT %QX0.7	:BOOL;	 (* 	SAFETY DOOR LOCK	*)

O_Weighing_CV_ON			AT %QX1.0	:BOOL;	 (* 	WEIGHING CONVEYOR STARTER OK	*)						
O_ER_BufCv_Mtr1_On			AT %QX1.1	:BOOL;	 (* 	CARTON CV MOTOR 1 ON	*)
O_ER_BufCv_Mtr2_On			AT %QX1.2	:BOOL;	 (* 	CARTON CV MOTOR 2 ON	*)
O_ER_BFlapL_Vac_On			AT %QX1.3	:BOOL;	 (* 	4Y1 - ERECTOR BOTTOM LEFT FLAP VACUUM VALVE ON	*)
O_ER_BFlapR_Vac_On			AT %QX1.4	:BOOL;	 (* 	5Y1 - ERECTOR BOTTOM RIGHT FLAP VACUUM VALVE ON	*)
O_ER_Arm_Vac_On				AT %QX1.5	:BOOL;	 (* 	6Y1 - ERECTOR ARM VACUUM VALVE ON	*)
O_Nord_ValveL_On			AT %QX1.6	:BOOL;	 (* 	NORDSON LEFT DISPENSE VALVE ON	*)
O_Nord_ValveR_On			AT %QX1.7	:BOOL;	 (* 	NORDSON RIGHT DISPENSE VALVE ON	*)

QW_41DO2					AT %QB2:WORD;												
O_TnT_CaseFormat			AT %QX2.0	:BOOL;	 (* 	Track and Trace Case Format	*)
O_TnT_CrossPushToCase		AT %QX2.1	:BOOL;	 (* 	Track and Trace Cross Push to Case Initiated	*)
O_TnT_CrossPushForward		AT %QX2.2	:BOOL;	 (* 	Track and Trace Cross Push Fully Forward	*)
O_TnT_CaseIndex				AT %QX2.3	:BOOL;	 (* 	Track and Trace Case Index	*)
O_TnT_GoodCaseDischarge		AT %QX2.4	:BOOL;	 (* 	Track and Trace Good Case Discharge	*)
QX25						AT %QX2.5	:BOOL;	 (* 	SPARE	*)
QX26						AT %QX2.6	:BOOL;	 (* 	SPARE	*)
QX27						AT %QX2.7	:BOOL;	 (* 	SPARE	*)

O_UpStream_ReqToStpNO		AT %QX3.0	:BOOL;	 (* 	UPSTREAM REQUEST TO STOP CLOSE=ACTIVE	*)						
O_UpStream_ReqToStpNC		AT %QX3.1	:BOOL;	 (* 	UPSTREAM MACHINE RUNNING OPEN=ACTIVE	*)
QX32						AT %QX3.2	:BOOL;	 (* 	SPARE	*)
O_UpStream_ReqEmptying		AT %QX3.3	:BOOL;	 (* 	UPSTREAM REQUEST EMPTYING	*)
O_DnStream_ReqToStpNO		AT %QX3.4	:BOOL;	 (* 	DOWNSTREAM REQUEST TO STOP OPEN=ACTIVE	*)
O_DnStream_ReqToStpNC		AT %QX3.5	:BOOL;	 (* 	DOWNSTREAM REQUEST RUNNING CLOSE=ACTIVE	*)
O_DnStream_Reject			AT %QX3.6	:BOOL;	 (* 	DOWNSTREAM REQUEST EMPTYING	*)
QX37						AT %QX3.7	:BOOL;	 (* 	SPARE	*)

(**************************************************************************)
(*Erector Field IO - 60A1*)
(*Erector Left Assembly - Carton Supply & Flap Close*)

IW_60A1				AT %IB10:WORD;						
I_ER_BufferL_PE		AT %IX10.0	:BOOL;	 (* 	ERECTOR CARTON BUFFER PRESENT (LEFT), OFF=CARTON PRESENT	*)
I_ER_EmptyL_PE		AT %IX10.1	:BOOL;	 (* 	ERECTOR CARTON BUFFER EMPTY (LEFT)	*)
I_ER_RefillL_PE		AT %IX10.2	:BOOL;	 (* 	ERECTOR CARTON BUFFER REFILL (LEFT)	*)
I_EX_StpL_Dn		AT %IX10.3	:BOOL;	 (* 	EXIT STOPPER DOWN (LEFT)	*)
I_ER_FFlapL_Fwd		AT %IX10.4	:BOOL;	 (* 	ERECTOR FRONT FLAP CLOSING CYL FWD RS (LEFT)	*)
I_ER_FFlapL_Bwd		AT %IX10.5	:BOOL;	 (* 	ERECTOR FRONT FLAP CLOSING CYL BWD RS (LEFT)	*)
I_ER_BFlapL_Fwd		AT %IX10.6	:BOOL;	 (* 	FLAP OPENING FORWARD BOTTOM	(LEFT)*)
I_ER_BFlapL_Bwd		AT %IX10.7	:BOOL;	 (* 	FLAP OPENING BACKWARD BOTTOM (LEFT)*)


(**************************************************************************)
(*Erector Field IO - 61A1 *)
(*Erector Left Assembly - Flap Holder & Stopper*)

IW_61A1				AT %IB11:WORD;		
I_ER_StpL_Up		AT %IX11.0	:BOOL;	 (* 	ERECTOR STOPPER CYL UP RS (LEFT)	*)
I_ER_StpL_Dn		AT %IX11.1	:BOOL;	 (* 	ERECTOR STOPPER CYL DN RS (LEFT)	*)
I_ER_CaseGuideL_Fwd	AT %IX11.2	:BOOL;	 (* 	ERECTOR LEFT CASE GUIDE FORWARD (LEFT)	*)	
I_ER_CaseGuideL_Bwd	AT %IX11.3	:BOOL;	 (* 	ERECTOR LEFT CASE GUIDE BACKWARD (LEFT)	*)	
I_ER_RFlapL_Fwd		AT %IX11.4	:BOOL;	 (* 	ERECTOR REAR FLAP CLOSE FORWARD (LEFT)	*)	
I_ER_RFlapL_Bwd		AT %IX11.5	:BOOL;	 (* 	ERECTOR REAR FLAP CLOSE BACKWARD (LEFT)	*)	
I_ER_BFlapL_VacSw	AT %IX11.6	:BOOL;	 (* 	ERECTOR BOTTOM FLAP HOLD VACUUM SWITCH (LEFT)	*)	
I_ER_StpL_Ctn_PE	AT %IX11.7	:BOOL;	 (* 	ERECTOR CARTON PRESENCE AT  STOPPER (LEFT)	*)


(**************************************************************************)
(*Erector Field IO - 62A1 *)
(*Erector Right Assembly - Carton Supply & Flap Close*)

IW_62A1					AT %IB12:WORD;						
I_ER_TFlapOpnL_Fwd		AT %IX12.0	:BOOL;	 (* 	ERECTOR TOP FLAP OPENING CYL FWD RS (LEFT)	*)
I_ER_TFlapOpnL_Bwd		AT %IX12.1	:BOOL;	 (* 	ERECTOR TOP FLAP OPENING CYL BWD RS (LEFT)	*)
I_ER_TFlapClsL_Fwd		AT %IX12.2	:BOOL;	 (* 	ERECTOR TOP FLAP CLOSING CYL FWD RS (LEFT)	*)
I_ER_TFlapClsL_Bwd		AT %IX12.3	:BOOL;	 (* 	ERECTOR TOP FLAP CLOSING CYL BWD RS (LEFT)	*)
I_ER_FlapHoldL_Fwd 		AT %IX12.4	:BOOL;	 (* 	EXIT FLAP HOLDER LEFT CYL FWD RS (FOR GLUE DISPENSING)	*)
I_ER_FlapHoldL_Bwd		AT %IX12.5	:BOOL;	 (* 	EXIT FLAP HOLDER LEFT CYL BWD RS (FOR GLUE DISPENSING)	*)
I_EX_SquarenessL_Fwd	AT %IX12.6	:BOOL;	 (* 	SQUARENESS CYL FWD RS (LEFT) 	*)
I_EX_SquarenessL_Bwd	AT %IX12.7	:BOOL;	 (* 	SQUARENESS CYL BWD RS (LEFT)	*)

(**************************************************************************)
(*Erector Field IO - 63A1 *)
(*Erector Right Assembly - Flap Holder & Stopper*)

IW_63A1				AT %IB13:WORD;		
I_ER_BufferR_PE		AT %IX13.0	:BOOL;	 (* 	ERECTOR CARTON BUFFER PRESENT (RIGHT), OFF=CARTON PRESENT	*)	
I_ER_EmptyR_PE		AT %IX13.1	:BOOL;	 (* 	ERECTOR CARTON BUFFER EMPTY (RIGHT)	*)
IX132				AT %IX13.2	:BOOL;	 (* 	SPARE	*)
I_EX_StpR_Dn		AT %IX13.3	:BOOL;	 (* 	EXIT STOPPER DOWN (RIGHT)	*)
I_ER_FFlapR_Fwd		AT %IX13.4	:BOOL;	 (* 	ERECTOR FRONT FLAP CLOSING CYL FWD RS (RIGHT)	*)
I_ER_FFlapR_Bwd		AT %IX13.5	:BOOL;	 (* 	ERECTOR FRONT FLAP CLOSING CYL BWD RS (RIGHT)	*)
I_ER_BFlapR_Fwd		AT %IX13.6	:BOOL;	 (* 	ERECTOR BOTTOM FLAP HOLD FWD RS (RIGHT)	*)
I_ER_BFlapR_Bwd		AT %IX13.7	:BOOL;	 (* 	ERECTOR BOTTOM FLAP HOLD BWD RS (RIGHT)	*)
				

(**************************************************************************)
(*Erector Field IO - 64A1 *)
(*Erector Right Assembly - Flap Holder & Stopper*)
IW_64A1				AT %IB14:WORD;	
I_ER_StpR_Up		AT %IX14.0	:BOOL;	 (* 	ERECTOR STOPPER CYL UP RS (RIGHT)	*)
I_ER_StpR_Dn		AT %IX14.1	:BOOL;	 (* 	ERECTOR STOPPER CYL DN RS (RIGHT)	*)
I_ER_CaseGuideR_Fwd	AT %IX14.2	:BOOL;	 (* 	ERECTOR LEFT CASE GUIDE FORWARD (RIGHT)	*)	
I_ER_CaseGuideR_Bwd	AT %IX14.3	:BOOL;	 (* 	ERECTOR LEFT CASE GUIDE BACKWARD (RIGHT)	*)	
I_ER_RFlapR_Fwd		AT %IX14.4	:BOOL;	 (* 	ERECTOR REAR FLAP CLOSING CYL FWD RS (RIGHT)	*)
I_ER_RFlapR_Bwd		AT %IX14.5	:BOOL;	 (* 	ERECTOR REAR FLAP CLOSING CYL BWD RS (RIGHT)	*)
I_ER_BFlapR_VacSw	AT %IX14.6	:BOOL;	 (* 	ERECTOR BOTTOM FLAP HOLD VACUUM SWITCH (RIGHT)	*)
I_ER_StpR_Ctn_PE	AT %IX14.7	:BOOL;	 (* 	ERECTOR CARTON PRESENCE AT  STOPPER (RIGHT)	*)


(**************************************************************************)
(*Erector Field IO - 65A1 *)
(*Erector Right Assembly - Flap Holder & Stopper*)
IW_65A1					AT %IB15:WORD;
I_ER_TFlapOpnR_Fwd		AT %IX15.0	:BOOL;	 (* 	ERECTOR TOP FLAP OPENING CYL FWD RS (RIGHT)	*)
I_ER_TFlapOpnR_Bwd		AT %IX15.1	:BOOL;	 (* 	ERECTOR TOP FLAP OPENING CYL BWD RS (RIGHT)	*)
I_ER_TFlapClsR_Fwd		AT %IX15.2	:BOOL;	 (* 	ERECTOR TOP FLAP CLOSING CYL FWD RS (RIGHT)	*)
I_ER_TFlapClsR_Bwd		AT %IX15.3	:BOOL;	 (* 	ERECTOR TOP FLAP CLOSING CYL BWD RS (RIGHT)	*)
I_ER_FlapHoldR_Fwd 		AT %IX15.4	:BOOL;	 (* 	EXIT FLAP HOLDER RIGHT CYL FWD RS (FOR GLUE DISPENSING)	*)
I_ER_FlapHoldR_Bwd		AT %IX15.5	:BOOL;	 (* 	EXIT FLAP HOLDER RIGHT CYL BWD RS (FOR GLUE DISPENSING)	*)
I_EX_SquarenessR_Fwd	AT %IX15.6	:BOOL;	 (* 	SQUARENESS CYL FWD RS (LEFT)	*)
I_EX_SquarenessR_Bwd	AT %IX15.7	:BOOL;	 (* 	SQUARENESS CYL BWD RS (LEFT)	*)


(**************************************************************************)
(*Erector Field IO - 66A1 *)
(*Erector Arm Assembly*)
IW_66A1					AT %IB16:WORD;
I_ER_ArmTilt_Fwd		AT %IX16.0	:BOOL;	 (* 	ERECTOR ARM TILT CYL FWD RS	*)
I_ER_ArmTilt_Bwd		AT %IX16.1	:BOOL;	 (* 	ERECTOR ARM TILT CYL BWD RS	*)
I_ER_Arm_Up				AT %IX16.2	:BOOL;	 (* 	ERECTOR ARM CYL UP RS	*)
I_ER_Arm_Dn				AT %IX16.3	:BOOL;	 (* 	ERECTOR ARM CYL DOWN RS	*)
IX164					AT %IX16.4	:BOOL;	 (* 	SPARE	*)
IX165					AT %IX16.5	:BOOL;	 (* 	SPARE	*)			
I_ER_Arm_VacSw			AT %IX16.6	:BOOL;	 (* 	ERECTOR ARM VACUUM SWITCH	*)
I_EX_Cv_Ctn_PE	 		AT %IX16.7	:BOOL;	 (* 	EXIT WEIGHT CHECKER PRODUCT PRESENCE SENSOR	*)




I_Weighing						AT %I*		: DINT;
I_Weighing_Status_SteadyBit		AT %I*		: BOOL;

END_VAR

// ---- GVLs/IO/GVL_Valve_Manifold.TcGVL
VAR_GLOBAL
	
(**************************************************************************)
(*Erector Valve Manifold - 70A1*)
QW_70A1						AT %QB50:WORD;
QW_70A1_0					AT %QB52:WORD;
QW_70A1_1					AT %QB50:BYTE;
QW_70A1_2					AT %QB51:BYTE;
QW_70A1_3					AT %QB52:BYTE;
QW_70A1_4					AT %QB53:BYTE;

O_ER_FFlapL_Fwd				AT %QX50.0	:BOOL;	 (* 	1Y1 - ERECTOR FRONT FLAP CLOSING CYL FWD SV (LEFT)	*)
O_ER_FFlapL_Bwd				AT %QX50.1	:BOOL;	 (* 	1Y1 - ERECTOR FRONT FLAP CLOSING CYL BWD SV (LEFT)	*)	
O_ER_BFlapL_Fwd				AT %QX50.2	:BOOL;	 (* 	1Y2 - ERECTOR BOTTOM FLAP HOLD FWD SV (LEFT)	*)
O_ER_BFlapL_Bwd				AT %QX50.3	:BOOL;	 (* 	1Y2 - ERECTOR BOTTOM FLAP HOLD BWD SV (LEFT)	*)
O_ER_StpL_Up				AT %QX50.4	:BOOL;	 (* 	1Y3 - ERECTOR STOPPER CYL UP SV (LEFT)	*)
O_ER_StpL_Dn				AT %QX50.5	:BOOL;	 (* 	1Y3 - ERECTOR STOPPER CYL DN SV (LEFT)	*)
O_ER_CaseGuideL_Fwd			AT %QX50.6	:BOOL;	 (* 	1Y4 - ERECTOR CASE GUIDE CYL FWD SV (LEFT)	*)
O_ER_CaseGuideL_Bwd			AT %QX50.7	:BOOL;	 (* 	1Y4 - ERECTOR CASE GUIDE CYL BWD SV (LEFT)	*)
O_ER_RFlapL_Fwd				AT %QX51.0	:BOOL;	 (* 	1Y5 - ERECTOR REAR FLAP CLOSING CYL FWD SV (LEFT)	*)
O_ER_RFlapL_Bwd				AT %QX51.1	:BOOL;	 (* 	1Y5 - ERECTOR REAR FLAP CLOSING CYL BWD SV (LEFT)	*)
O_ER_TFlapOpnL_Fwd			AT %QX51.2	:BOOL;	 (* 	1Y6 - ERECTOR TOP FLAP OPENING CYL FWD SV (LEFT)	*)
O_ER_TFlapOpnL_Bwd			AT %QX51.3	:BOOL;	 (* 	1Y6 - ERECTOR TOP FLAP OPENING CYL BWD SV (LEFT)	*)
O_ER_TFlapClsL_Fwd			AT %QX51.4	:BOOL;	 (* 	1Y7 - ERECTOR TOP FLAP CLOSING CYL FWD SV (LEFT)	*)
O_ER_TFlapClsL_Bwd			AT %QX51.5	:BOOL;	 (* 	1Y7 - ERECTOR TOP FLAP CLOSING CYL BWD SV (LEFT)	*)
O_ER_FlapHoldL_Fwd			AT %QX51.6	:BOOL;	 (* 	1Y8 - EXIT FLAP HOLDER LEFT CYL FWD SV (FOR GLUE DISPENSING)	*)
O_ER_FlapHoldL_Bwd			AT %QX51.7	:BOOL;	 (* 	1Y8 - EXIT FLAP HOLDER LEFT CYL BWD SV (FOR GLUE DISPENSING)	*)
O_ER_ArmTilt_Fwd			AT %QX52.0	:BOOL;	 (* 	1Y9 - ERECTOR ARM TILT CYL FWD SV	*)
O_ER_ArmTilt_Bwd			AT %QX52.1	:BOOL;	 (* 	1Y9 - ERECTOR ARM TILT CYL BWD SV	*)
O_ER_Arm_Up					AT %QX52.2	:BOOL;	 (* 	1Y10 - ERECTOR ARM CYL UP SV	*)
O_ER_Arm_Dn					AT %QX52.3	:BOOL;	 (* 	1Y10 - ERECTOR ARM CYL DOWN SV	*)
O_EX_SquarenessCylL_Fwd		AT %QX52.4	:BOOL;	 (* 	1Y11 - SQUARENESS CYLINDER FORWARD (LEFT)	*)
O_EX_SquarenessCylL_Bwd		AT %QX52.5	:BOOL;	 (* 	1Y11 - SQUARENESS CYLINDER BACKWARD (LEFT)	*)
O_EX_StpCylL_Up				AT %QX52.6	:BOOL;	 (* 	1Y12 - EXIT STOPPER CYLINDER UP (LEFT)	*)
O_EX_StpCylL_Dn				AT %QX52.7	:BOOL;	 (* 	1Y12 - EXIT STOPPER CYLINDER DOWN (LEFT)	*)

	
(**************************************************************************)
(*Erector Valve Manifold - 71A1*)
QW_71A1						AT %QB60:WORD;
QW_71A1_1					AT %QB60:BYTE;
QW_71A1_2					AT %QB61:BYTE;
QW_71A1_3					AT %QB62:BYTE;
QW_71A1_4					AT %QB63:BYTE;

O_ER_FFlapR_Fwd				AT %QX60.0	:BOOL;	 (* 	2Y1 - ERECTOR FRONT FLAP CLOSING CYL FWD SV (RIGHT)	*)
O_ER_FFlapR_Bwd				AT %QX60.1	:BOOL;	 (* 	2Y1 - ERECTOR FRONT FLAP CLOSING CYL BWD SV (RIGHT)	*)	
O_ER_BFlapR_Fwd				AT %QX60.2	:BOOL;	 (* 	2Y2 - ERECTOR BOTTOM FLAP HOLD FWD SV (RIGHT)	*)
O_ER_BFlapR_Bwd				AT %QX60.3	:BOOL;	 (* 	2Y2 - ERECTOR BOTTOM FLAP HOLD BWD SV (RIGHT)	*)
O_ER_StpR_Up				AT %QX60.4	:BOOL;	 (* 	2Y3 - ERECTOR STOPPER CYL UP SV (RIGHT)	*)
O_ER_StpR_Dn				AT %QX60.5	:BOOL;	 (* 	2Y3 - ERECTOR STOPPER CYL DN SV (RIGHT)	*)
O_ER_CaseGuideR_Fwd			AT %QX60.6	:BOOL;	 (* 	2Y4 - ERECTOR CASE GUIDE CYL FWD SV (RIGHT)	*)
O_ER_CaseGuideR_Bwd			AT %QX60.7	:BOOL;	 (* 	2Y4 - ERECTOR CASE GUIDE CYL BWD SV (RIGHT)	*)
O_ER_RFlapR_Fwd				AT %QX61.0	:BOOL;	 (* 	2Y5 - ERECTOR REAR FLAP CLOSING CYL FWD SV (RIGHT)	*)
O_ER_RFlapR_Bwd				AT %QX61.1	:BOOL;	 (* 	2Y5 - ERECTOR REAR FLAP CLOSING CYL BWD SV (RIGHT)	*)
O_ER_TFlapOpnR_Fwd			AT %QX61.2	:BOOL;	 (* 	2Y6 - ERECTOR TOP FLAP OPENING CYL FWD SV (RIGHT)	*)
O_ER_TFlapOpnR_Bwd			AT %QX61.3	:BOOL;	 (* 	2Y6 - ERECTOR TOP FLAP OPENING CYL BWD SV (RIGHT)	*)
O_ER_TFlapClsR_Fwd			AT %QX61.4	:BOOL;	 (* 	2Y7 - ERECTOR TOP FLAP CLOSING CYL FWD SV (RIGHT)	*)
O_ER_TFlapClsR_Bwd			AT %QX61.5	:BOOL;	 (* 	2Y7 - ERECTOR TOP FLAP CLOSING CYL BWD SV (RIGHT)	*)
O_EX_FlapHoldR_Fwd			AT %QX61.6	:BOOL;	 (* 	2Y8 - EXIT FLAP HOLDER RIGHT CYL FWD SV (FOR GLUE DISPENSING)	*)
O_EX_FlapHoldR_Bwd			AT %QX61.7	:BOOL;	 (* 	2Y8 - EXIT FLAP HOLDER RIGHT CYL BWD SV (FOR GLUE DISPENSING)	*)
O_EX_SquarenessCylR_Fwd		AT %QX62.0	:BOOL;	 (* 	2Y9 - SQUARENESS CYLINDER FORWARD (RIGHT)	*)
O_EX_SquarenessCylR_Bwd		AT %QX62.1	:BOOL;	 (* 	2Y9 - SQUARENESS CYLINDER BACKWARD (RIGHT)	*)
O_EX_StpCylR_Up				AT %QX62.2	:BOOL;	 (* 	2Y10 - EXIT STOPPER CYLINDER UP (RIGHT)	*)
O_EX_StpCylR_Dn				AT %QX62.3	:BOOL;	 (* 	2Y10 - EXIT STOPPER CYLINDER DOWN (RIGHT)	*)

(**************************************************************************)
(*Collator Valve Manifold - 170A1*)

QW_170A1				AT %QB150:WORD;
QW_170A1_1				AT %QB150:BYTE;
QW_170A1_2				AT %QB151:BYTE;

O_CO_YPush_Dn			AT %QX150.0	:BOOL;	 (* 	3Y1 - COLLATOR X-PUSHER DOWN	*)
O_CO_YPush_Up			AT %QX150.1	:BOOL;	 (* 	3Y1 - COLLATOR X-PUSHER UP	*)
O_CO_YPush_Strk_Fwd		AT %QX150.2	:BOOL;	 (* 	3Y2 - COLLATOR Y PUSHER STROKE CYL FWD SV	*)
O_CO_YPush_Strk_Bwd		AT %QX150.3	:BOOL;	 (* 	3Y2 - COLLATOR Y PUSHER STROKE CYL BWD SV	*)
O_CO_Brdg_Fwd			AT %QX150.4	:BOOL;	 (* 	3Y3 - COLLATOR PUSHER BRIDGE CYL FWD SV	*)
O_CO_Brdg_Bwd			AT %QX150.5	:BOOL;	 (* 	3Y3 - COLLATOR PUSHER BRIDGE CYL BWD SV	*)
O_CO_RFlapGuide_Fwd		AT %QX150.6	:BOOL;	 (* 	3Y5 - COLLATOR PUSHER REAR GUIDE FLAP BRIDGE CYL FWD SV	*)
O_CO_RFlapGuide_Bwd		AT %QX150.7	:BOOL;	 (* 	3Y5 - COLLATOR PUSHER REAR GUIDE FLAP BRIDGE CYL BWD SV	*)
O_CO_FFlapBrdg_Fwd		AT %QX151.0	:BOOL;	 (* 	3Y4 - COLLATOR PUSHER FRONT GUIDE FLAP BRIDGE CYL FWD SV	*)
O_CO_FFlapBrdg_Bwd		AT %QX151.1	:BOOL;	 (* 	3Y4 - COLLATOR PUSHER FRONT GUIDE FLAP BRIDGE CYL BWD SV	*)
O_CO_PalletLocating_Fwd	AT %QX151.2 :BOOL;
O_CO_PalletLocating_Bwd	AT %QX151.3 :BOOL;
O_CO_Sing1_Fwd			AT %QX151.4 :BOOL;
O_CO_Sing1_Bwd			AT %QX151.5 :BOOL;
O_CO_Sing2_Fwd			AT %QX151.6 :BOOL;
O_CO_Sing2_Bwd			AT %QX151.7 :BOOL;

(**************************************************************************)
(*Exit Valve Manifold - 350A1*)

QW_350A1				AT %QB350:WORD;
QB350A1_1				AT %QB350:BYTE;
QB350A1_2				AT %QB351:BYTE;

O_EL_TapeOpening_Fwd	AT %QX350.0	:BOOL;	 (* 	4Y1 - VERTICAL TAPE OPENING CYL FWD SV	*)
O_EL_TapeOpening_Bwd	AT %QX350.1	:BOOL;	 (* 	4Y1 - VERTICAL TAPE OPENING CYL BWD SV	*)
O_EL_TiltLift_Fwd		AT %QX350.2	:BOOL;	 (* 	4Y2 - VERTICAL EXIT TILT LIFT CYL FWD SV	*)
O_EL_TiltLift_Bwd		AT %QX350.3	:BOOL;	 (* 	4Y2 - VERTICAL EXIT TILT LIFT CYL BWD SV	*)
O_EL_TapeLock_ON		AT %QX350.4	:BOOL;	 (* 	4Y3 - VERTICAL WA TAPE LOCK ACTIVE SV	*)
O_EL_TiltVacLift_Up		AT %QX350.6	:BOOL;	 (* 	4Y4 - VERTICAL EXIT TILT VACUUM LIFT CYL UP SV	*)
O_EL_TiltVacLift_Dn		AT %QX350.7	:BOOL;	 (* 	4Y4 - VERTICAL EXIT TILT VACUUM LIFT CYL DN SV	*)
O_EL_TapeChange_Fwd		AT %QX351.0	:BOOL;	 (* 	4Y5 - VERTICAL TAPE CHANGE CYL FWD SV	*)
O_EL_TapeChange_Bwd		AT %QX351.1	:BOOL;	 (* 	4Y5 - VERTICAL TAPE CHANGE CYL BWD SV	*)
						
















O_ER_BFlapCloseL_Fwd		AT %QX950.0	:BOOL;	 (* 	1Y1 - ERECTOR BOTTOM FLAP CLOSE FWD SV (LEFT)	*)
O_ER_BFlapCloseL_Bwd		AT %QX950.1	:BOOL;	 (* 	1Y1 - ERECTOR BOTTOM FLAP CLOSE BWD SV (LEFT)	*)
					
O_ER_BFlapCloseR_Fwd		AT %QX952.0	:BOOL;	 (* 	1Y9 - ERECTOR BOTTOM FLAP CLOSE FWD SV (RIGHT)	*)
O_ER_BFlapCloseR_Bwd		AT %QX952.1	:BOOL;	 (* 	1Y9 - ERECTOR BOTTOM FLAP CLOSE BWD SV (RIGHT)	*)

O_CO_StkRel_Fwd		AT %QX150.2	:BOOL;	 (* 	2Y2 - COLLATOR STACK RELEASE CYLINDER FWD SV	*)
O_CO_StkRel_Bwd		AT %QX150.3	:BOOL;	 (* 	2Y2 - COLLATOR STACK RELEASE CYLINDER BWD SV	*)








END_VAR

// ---- GVLs/MC/GVL_General.TcGVL
{attribute 'Tc2GvlVarNames'}
VAR_GLOBAL
(**************************************************************************************************************)
(* System Bit *)
(**************************************************************************************************************)

	OFF_50ms		: BOOL;
	ON_50ms			: BOOL;
	Clock50msOnPls	: BOOL;
	OFF_100ms		: BOOL;
	ON_100ms		: BOOL;
	Clock100msOnPls	: BOOL;
	OFF_500ms		: BOOL;
	ON_500ms		: BOOL;
	Clock500msOnPls	: BOOL;
	OFF_1s			: BOOL;
	ON_1s			: BOOL;
	Clock1sOnPls	: BOOL;
	Always_ON		: BOOL;
	Always_Off		: BOOL;
	Debug			: BOOL := TRUE;
	TestSequence	: BOOL;

	
(**************************************************************************************************************)
(* Machine Standard Word *)
(**************************************************************************************************************)

	ErrorDWord 			AT %MB1000:  ARRAY [0..20,1..10] OF DWORD;
	WarningDWord		AT %MB2000: ARRAY [0..20,1..10] OF DWORD;
	AutoDWord 			AT %MB3000:  ARRAY [0..20,1..10] OF DWORD;
	OriginDWord 		AT %MB4000:  ARRAY [0..20,1..10] OF DWORD;

	InputByte			AT %IB0: ARRAY [0..500] OF BYTE;
	OutputByte			AT %QB0: ARRAY [0..500] OF BYTE;

(**************************************************************************************************************)
(* Machine and Station Control *)
(**************************************************************************************************************)
	MC:structMachineCtrl;
	MC_Ctrl:fbMachineCtrl;

	SC :ARRAY[0..6] OF structStationCtrl;
	
	CO	:structStationCtrl;				(*Structure only used for display and read only*)
	CO_Stack :structStationCtrl;		(*Structure only used for display and read only*)
	CO_XPush :structStationCtrl;		(*Structure only used for display and read only*)
	CO_YPush :structStationCtrl;		(*Structure only used for display and read only*)
	ER	:structStationCtrl;				(*Structure only used for display and read only*)
	EX	:structStationCtrl;				(*Structure only used for display and read only*)
	EL	:structStationCtrl;				(*Structure only used for display and read only*)
	HOR	:structStationCtrl;				(*Structure only used for display and read only*)
	ER_FixedFlap :structStationCtrl;	(*Structure only used for display and read only*)
	
(**************************************************************************************************************)
(* Manual Control *)
(**************************************************************************************************************)
	ManualSafetyOK		:BOOL;
	M_StepFwdPls		:BOOL;
	M_StepBwdPls		:BOOL;
	M_StepRun			:BOOL;

(**************************************************************************************************************)
(* Input/Output *)
(**************************************************************************************************************)
	(*InputWord			AT%IB0	:ARRAY [0..100] OF BOOL;*)

(**************************************************************************************************************)
(* Light Curtain Muting Control *)
(**************************************************************************************************************)

	HOR_LC_Muting	:BOOL;	(*Control Bit to mute Horizontal light curtain*)
	EL_LC_Muting	:BOOL;	(*Control Bit to mute Elevator light curtain*)

(**************************************************************************************************************)
(* To Bypass The Erector Safety Sensor *)
(**************************************************************************************************************)	
	Erector_SafetySensorBypass	:BOOL;
	
END_VAR

VAR_GLOBAL CONSTANT

	Number_of_Station:INT:=6;	(*Note: SC Array Dimension cannot be smaller than this value*)	

END_VAR

// ---- GVLs/MC/GVL_Auto.TcGVL
{attribute 'Tc2GvlVarNames'}
VAR_GLOBAL

	A_EL_LC_Muting:bool; 	(*Mute Elevator Light Curtain in Auto*)
	A_AutorunDataOK:BOOL;	(*Recipe Data OK for Autorun to start*)
	
	A_HOR_LC_Muting:BOOL; 	(*Mute Horizontal Light Curtain in Auto*)
	
	
(**************************************************************************************************************)
(*----------   P0 - COLLATOR   ----------*)
(* All P0 control bits and words must be within address MD3000~MD3039*)
(* All bits and words within the address will be reset when not in autorun mode*)
(**************************************************************************************************************)
	A0_RunStep				AT %MW3000:INT;

